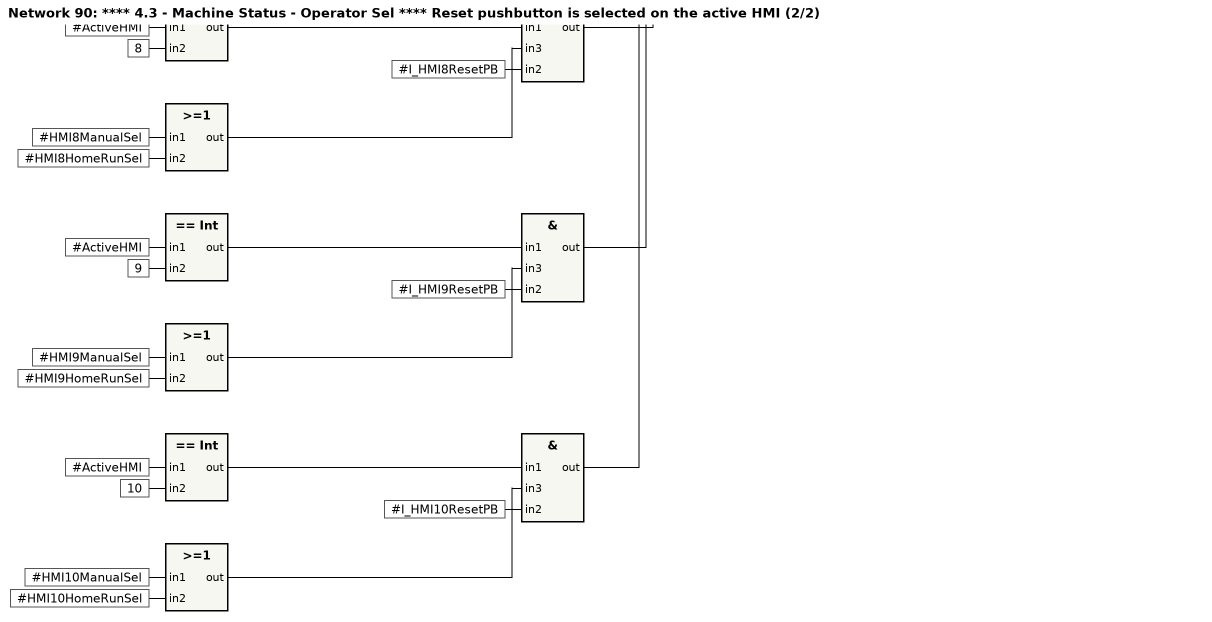
   #O_PBResetSel := (((#ActiveHMI = 1) AND (#HMI1ManualSel OR #HMI1HomeRunSel) AND #I_HMI1ResetPB) OR ((#ActiveHMI = 2) AND (#HMI2ManualSel OR #HMI2HomeRunSel) AND #I_HMI2ResetPB) OR ((#ActiveHMI = 3) AND (#HMI3ManualSel OR #HMI3HomeRunSel) AND #I_HMI3ResetPB) OR ((#ActiveHMI = 4) AND (#HMI4ManualSel OR #HMI4HomeRunSel) AND #I_HMI4ResetPB) OR ((#ActiveHMI = 5) AND (#HMI5ManualSel OR #HMI5HomeRunSel) AND #I_HMI5ResetPB) OR ((#ActiveHMI = 6) AND (#HMI6ManualSel OR #HMI6HomeRunSel) AND #I_HMI6ResetPB) OR ((#ActiveHMI = 7) AND (#HMI7ManualSel OR #HMI7HomeRunSel) AND #I_HMI7ResetPB) OR ((#ActiveHMI = 8) AND (#HMI8ManualSel OR #HMI8HomeRunSel) AND #I_HMI8ResetPB) OR ((#ActiveHMI = 9) AND (#HMI9ManualSel OR #HMI9HomeRunSel) AND #I_HMI9ResetPB) OR ((#ActiveHMI = 10) AND (#HMI10ManualSel OR #HMI10HomeRunSel) AND #I_HMI10ResetPB)) AND NOT #AllHmiAutoSel;
   #PBResetSel := #O_PBResetSel;
   #IO_Modes.LModeSelector.PBResetSel := #O_PBResetSel;
END_REGION

REGION Network 91: **** 4.3 - Machine Status - Operator Sel **** Homerun Redo is selected
   // Homerun Redo is selected
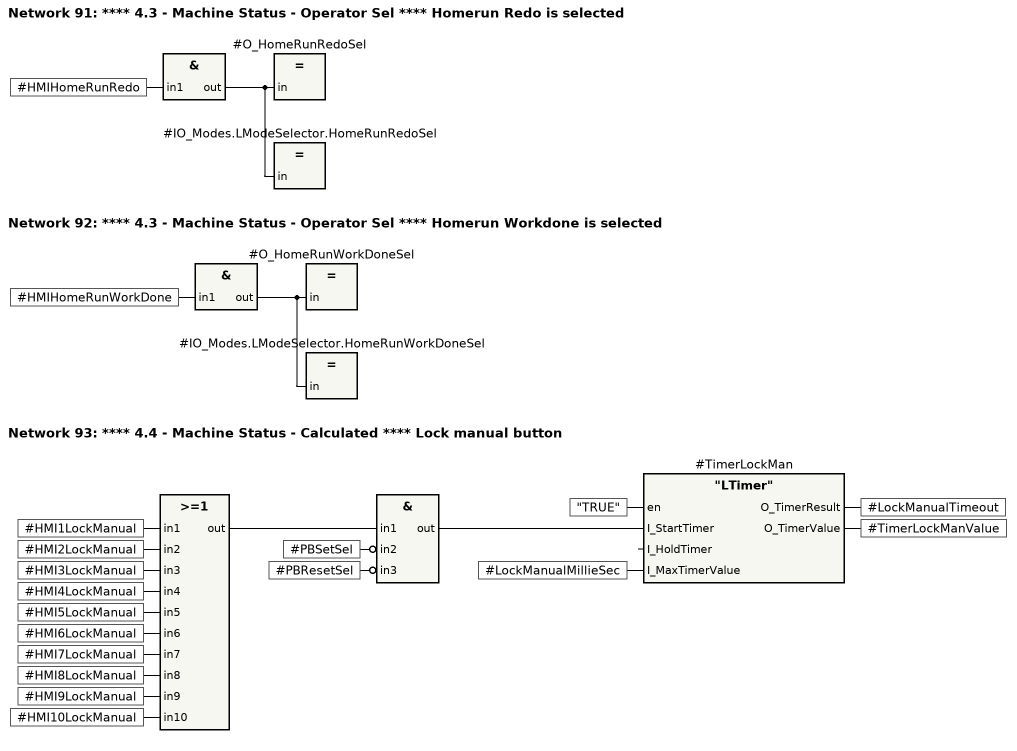
   #O_HomeRunRedoSel := #HMIHomeRunRedo;
   #IO_Modes.LModeSelector.HomeRunRedoSel := #HMIHomeRunRedo;
END_REGION

REGION Network 92: **** 4.3 - Machine Status - Operator Sel **** Homerun Workdone is selected
   // Homerun Workdone is selected
   #O_HomeRunWorkDoneSel := #HMIHomeRunWorkDone;
   #IO_Modes.LModeSelector.HomeRunWorkDoneSel := #HMIHomeRunWorkDone;
END_REGION

REGION Network 93: **** 4.4 - Machine Status - Calculated **** Lock manual button
   // Lock manual button
   IF "TRUE" THEN
       #TimerLockMan(I_StartTimer := (#HMI1LockManual OR #HMI2LockManual OR #HMI3LockManual OR #HMI4LockManual OR #HMI5LockManual OR #HMI6LockManual OR #HMI7LockManual OR #HMI8LockManual OR #HMI9LockManual OR #HMI10LockManual) AND NOT #PBSetSel AND NOT #PBResetSel,   // "LTimer"
                     I_MaxTimerValue := #LockManualMillieSec,
                     O_TimerResult => #LockManualTimeout,
                     O_TimerValue => #TimerLockManValue);
   END_IF;
END_REGION

REGION Network 94: **** 4.5 - Machine Status - Modes **** Auto is selected on all HMI
   // Auto is selected on all HMI
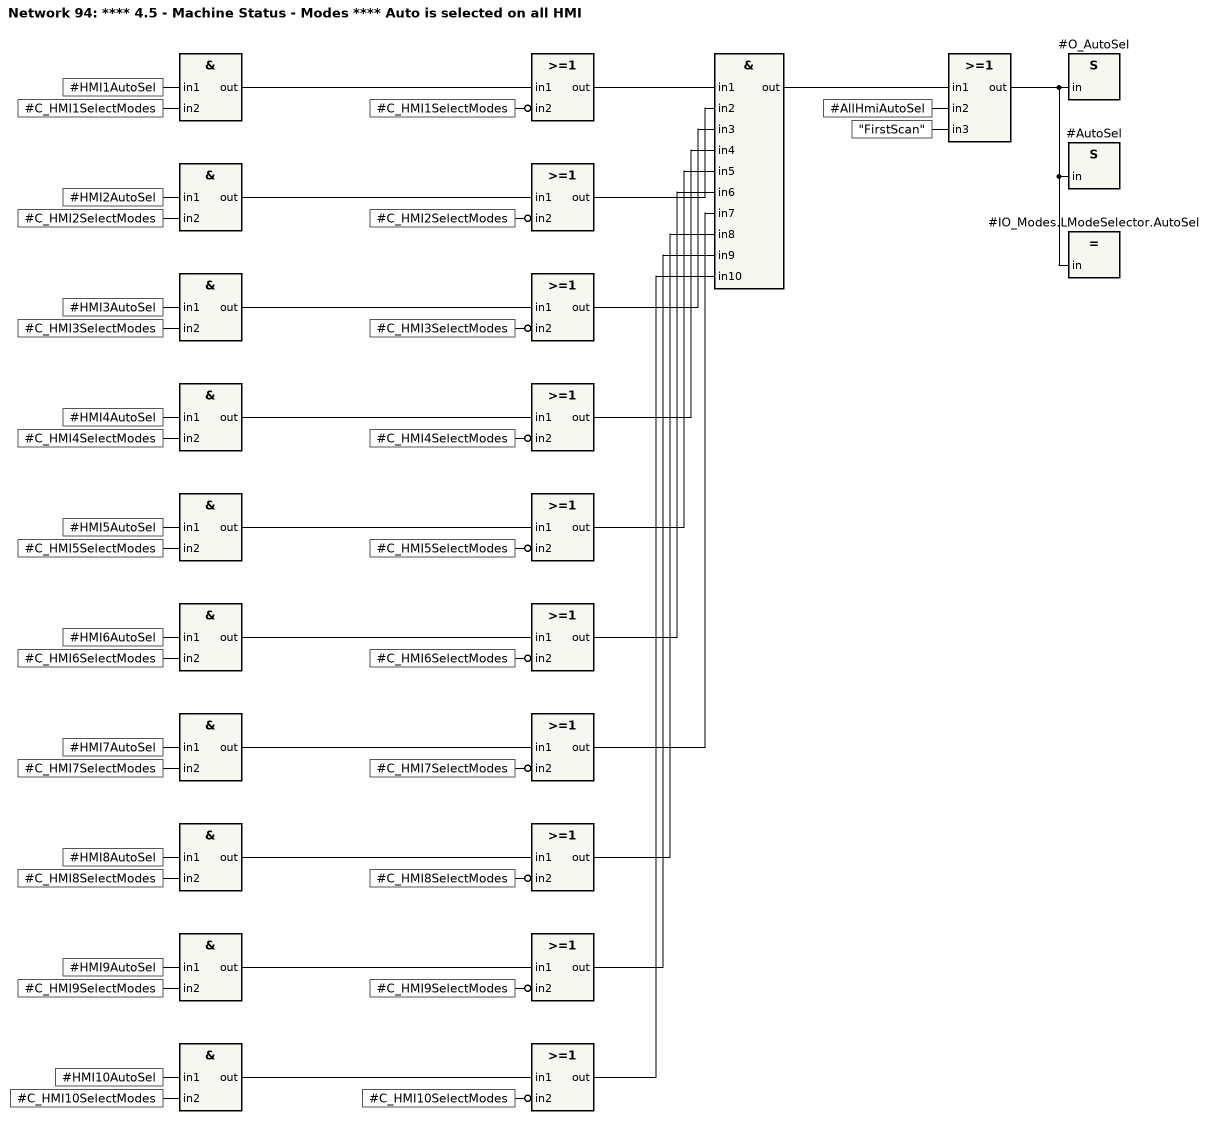
   #_w1 := (((#HMI1AutoSel AND #C_HMI1SelectModes) OR NOT #C_HMI1SelectModes) AND ((#HMI2AutoSel AND #C_HMI2SelectModes) OR NOT #C_HMI2SelectModes) AND ((#HMI3AutoSel AND #C_HMI3SelectModes) OR NOT #C_HMI3SelectModes) AND ((#HMI4AutoSel AND #C_HMI4SelectModes) OR NOT #C_HMI4SelectModes) AND ((#HMI5AutoSel AND #C_HMI5SelectModes) OR NOT #C_HMI5SelectModes) AND ((#HMI6AutoSel AND #C_HMI6SelectModes) OR NOT #C_HMI6SelectModes) AND ((#HMI7AutoSel AND #C_HMI7SelectModes) OR NOT #C_HMI7SelectModes) AND ((#HMI8AutoSel AND #C_HMI8SelectModes) OR NOT #C_HMI8SelectModes) AND ((#HMI9AutoSel AND #C_HMI9SelectModes) OR NOT #C_HMI9SelectModes) AND ((#HMI10AutoSel AND #C_HMI10SelectModes) OR NOT #C_HMI10SelectModes)) OR #AllHmiAutoSel OR "FirstScan";
   IF #_w1 THEN
       #O_AutoSel := TRUE;
       #AutoSel := TRUE;
   END_IF;
   #IO_Modes.LModeSelector.AutoSel := #_w1;
END_REGION

REGION Network 95: **** 4.5 - Machine Status - Modes **** Reset Auto is selected on all HMI
   // Reset Auto is selected on all HMI
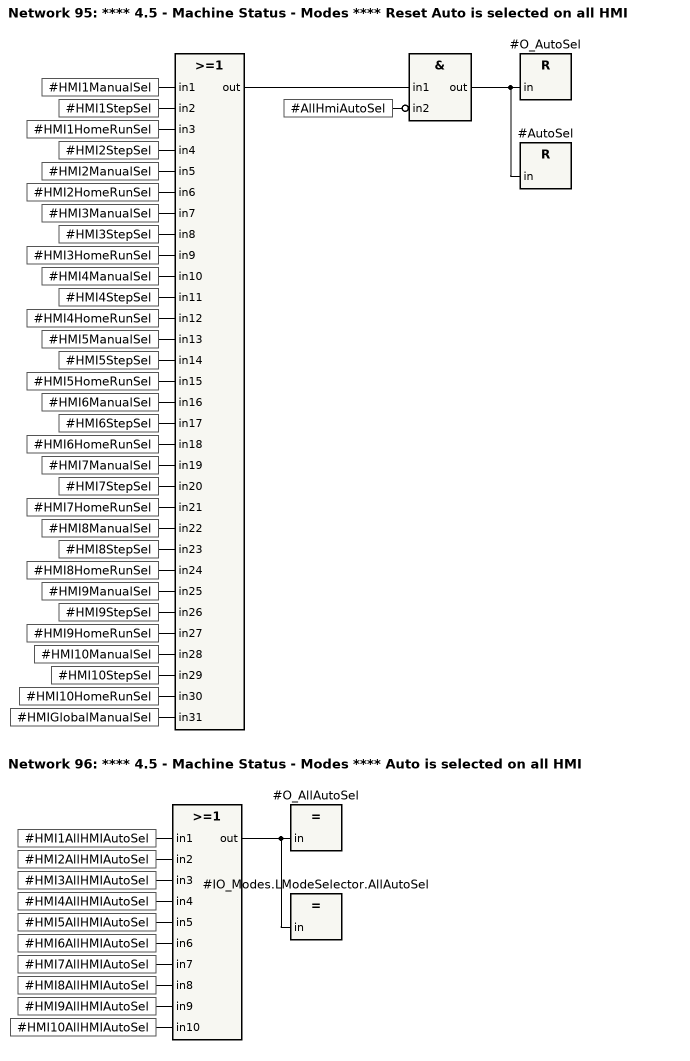
   IF (#HMI1ManualSel OR #HMI1StepSel OR #HMI1HomeRunSel OR #HMI2StepSel OR #HMI2ManualSel OR #HMI2HomeRunSel OR #HMI3ManualSel OR #HMI3StepSel OR #HMI3HomeRunSel OR #HMI4ManualSel OR #HMI4StepSel OR #HMI4HomeRunSel OR #HMI5ManualSel OR #HMI5StepSel OR #HMI5HomeRunSel OR #HMI6ManualSel OR #HMI6StepSel OR #HMI6HomeRunSel OR #HMI7ManualSel OR #HMI7StepSel OR #HMI7HomeRunSel OR #HMI8ManualSel OR #HMI8StepSel OR #HMI8HomeRunSel OR #HMI9ManualSel OR #HMI9StepSel OR #HMI9HomeRunSel OR #HMI10ManualSel OR #HMI10StepSel OR #HMI10HomeRunSel OR #HMIGlobalManualSel) AND NOT #AllHmiAutoSel THEN
       #O_AutoSel := FALSE;
       #AutoSel := FALSE;
   END_IF;
END_REGION

REGION Network 96: **** 4.5 - Machine Status - Modes **** Auto is selected on all HMI
   // Auto is selected on all HMI
   #O_AllAutoSel := #HMI1AllHMIAutoSel OR #HMI2AllHMIAutoSel OR #HMI3AllHMIAutoSel OR #HMI4AllHMIAutoSel OR #HMI5AllHMIAutoSel OR #HMI6AllHMIAutoSel OR #HMI7AllHMIAutoSel OR #HMI8AllHMIAutoSel OR #HMI9AllHMIAutoSel OR #HMI10AllHMIAutoSel;
   #IO_Modes.LModeSelector.AllAutoSel := #O_AllAutoSel;
END_REGION

REGION Network 97: **** 4.5 - Machine Status - Modes **** Step is selected on one HMI
   // Step is selected on one HMI
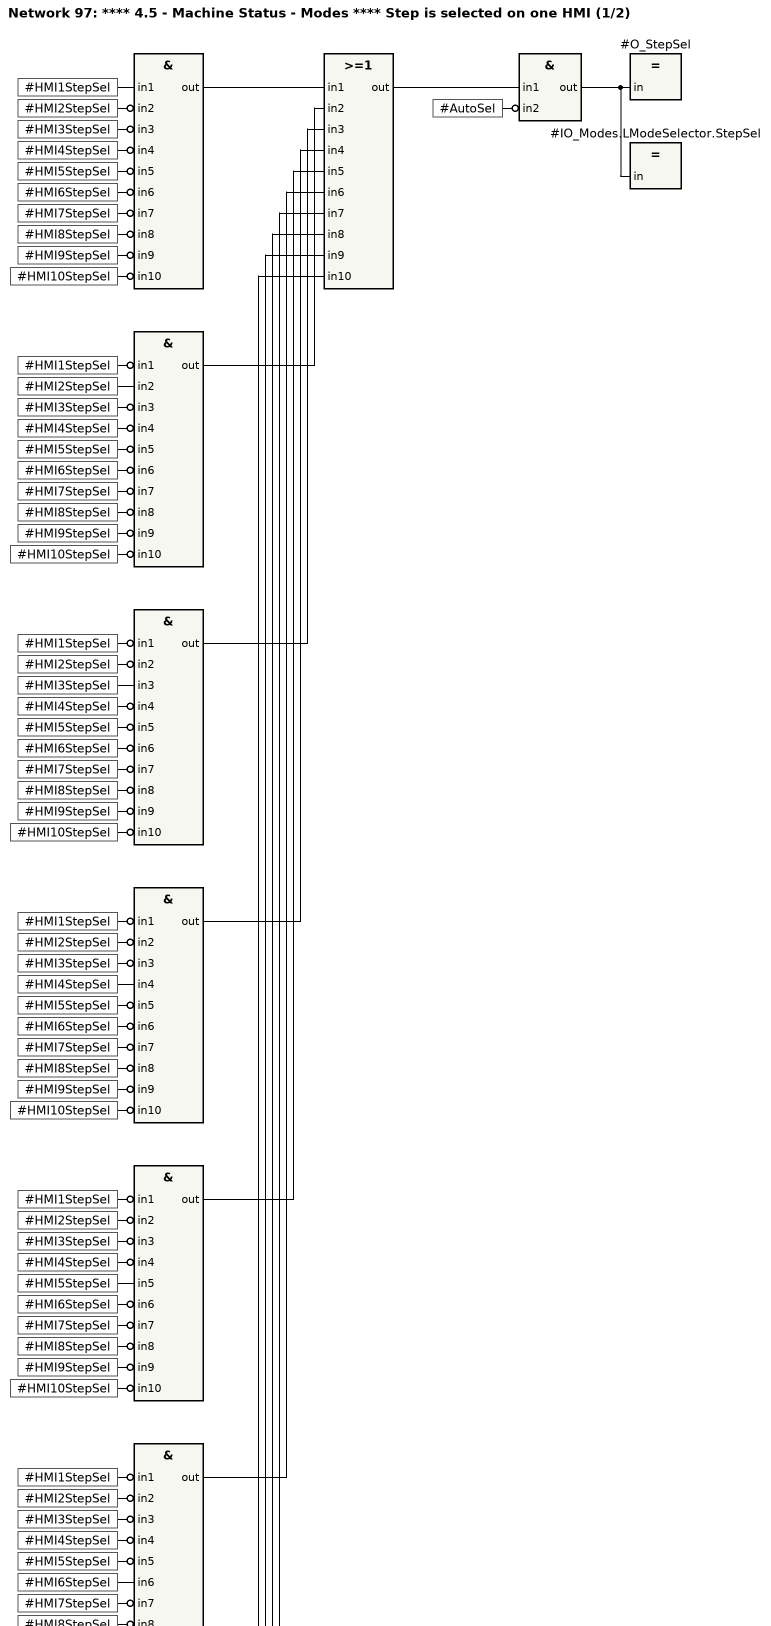
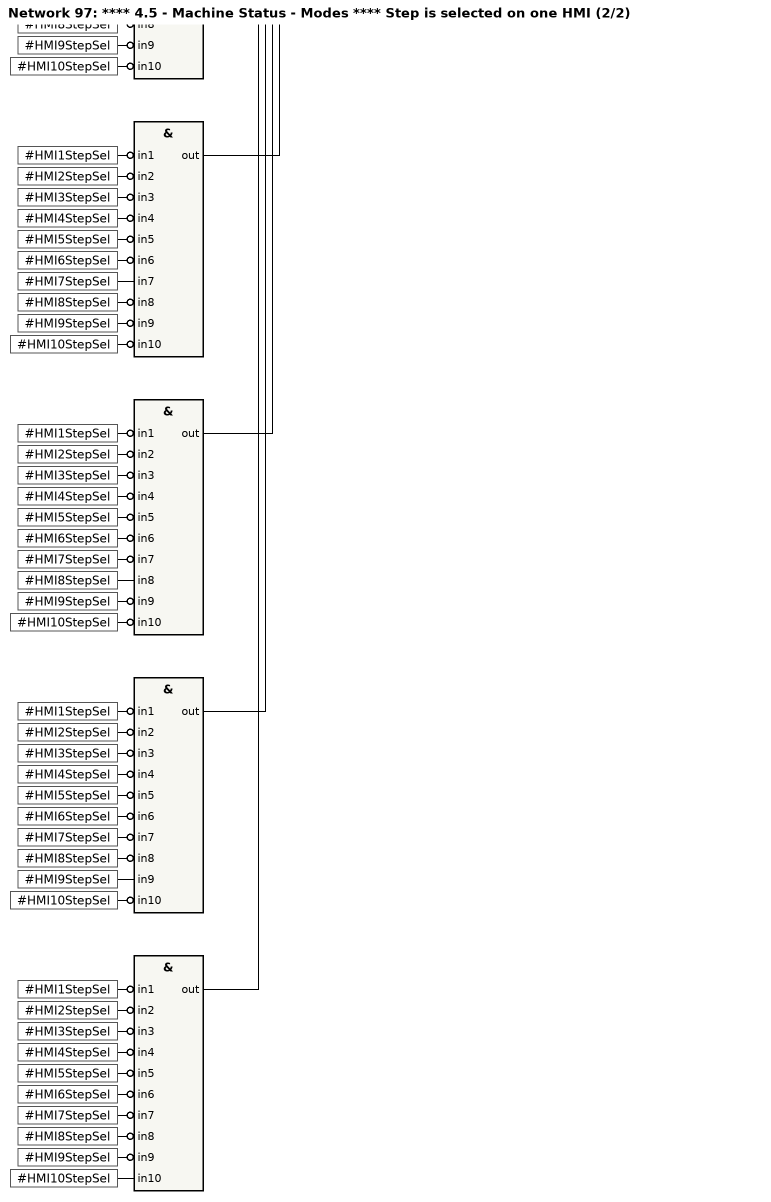
   #O_StepSel := ((#HMI1StepSel AND NOT #HMI2StepSel AND NOT #HMI3StepSel AND NOT #HMI4StepSel AND NOT #HMI5StepSel AND NOT #HMI6StepSel AND NOT #HMI7StepSel AND NOT #HMI8StepSel AND NOT #HMI9StepSel AND NOT #HMI10StepSel) OR (NOT #HMI1StepSel AND #HMI2StepSel AND NOT #HMI3StepSel AND NOT #HMI4StepSel AND NOT #HMI5StepSel AND NOT #HMI6StepSel AND NOT #HMI7StepSel AND NOT #HMI8StepSel AND NOT #HMI9StepSel AND NOT #HMI10StepSel) OR (NOT #HMI1StepSel AND NOT #HMI2StepSel AND #HMI3StepSel AND NOT #HMI4StepSel AND NOT #HMI5StepSel AND NOT #HMI6StepSel AND NOT #HMI7StepSel AND NOT #HMI8StepSel AND NOT #HMI9StepSel AND NOT #HMI10StepSel) OR (NOT #HMI1StepSel AND NOT #HMI2StepSel AND NOT #HMI3StepSel AND #HMI4StepSel AND NOT #HMI5StepSel AND NOT #HMI6StepSel AND NOT #HMI7StepSel AND NOT #HMI8StepSel AND NOT #HMI9StepSel AND NOT #HMI10StepSel) OR (NOT #HMI1StepSel AND NOT #HMI2StepSel AND NOT #HMI3StepSel AND NOT #HMI4StepSel AND #HMI5StepSel AND NOT #HMI6StepSel AND NOT #HMI7StepSel AND NOT #HMI8StepSel AND NOT #HMI9StepSel AND NOT #HMI10StepSel) OR (NOT #HMI1StepSel AND NOT #HMI2StepSel AND NOT #HMI3StepSel AND NOT #HMI4StepSel AND NOT #HMI5StepSel AND #HMI6StepSel AND NOT #HMI7StepSel AND NOT #HMI8StepSel AND NOT #HMI9StepSel AND NOT #HMI10StepSel) OR (NOT #HMI1StepSel AND NOT #HMI2StepSel AND NOT #HMI3StepSel AND NOT #HMI4StepSel AND NOT #HMI5StepSel AND NOT #HMI6StepSel AND #HMI7StepSel AND NOT #HMI8StepSel AND NOT #HMI9StepSel AND NOT #HMI10StepSel) OR (NOT #HMI1StepSel AND NOT #HMI2StepSel AND NOT #HMI3StepSel AND NOT #HMI4StepSel AND NOT #HMI5StepSel AND NOT #HMI6StepSel AND NOT #HMI7StepSel AND #HMI8StepSel AND NOT #HMI9StepSel AND NOT #HMI10StepSel) OR (NOT #HMI1StepSel AND NOT #HMI2StepSel AND NOT #HMI3StepSel AND NOT #HMI4StepSel AND NOT #HMI5StepSel AND NOT #HMI6StepSel AND NOT #HMI7StepSel AND NOT #HMI8StepSel AND #HMI9StepSel AND NOT #HMI10StepSel) OR (NOT #HMI1StepSel AND NOT #HMI2StepSel AND NOT #HMI3StepSel AND NOT #HMI4StepSel AND NOT #HMI5StepSel AND NOT #HMI6StepSel AND NOT #HMI7StepSel AND NOT #HMI8StepSel AND NOT #HMI9StepSel AND #HMI10StepSel)) AND NOT #AutoSel;
   #IO_Modes.LModeSelector.StepSel := #O_StepSel;
END_REGION

REGION Network 98: **** 4.5 - Machine Status - Modes **** Homerun is selected on one HMI
   // Homerun is selected on one HMI
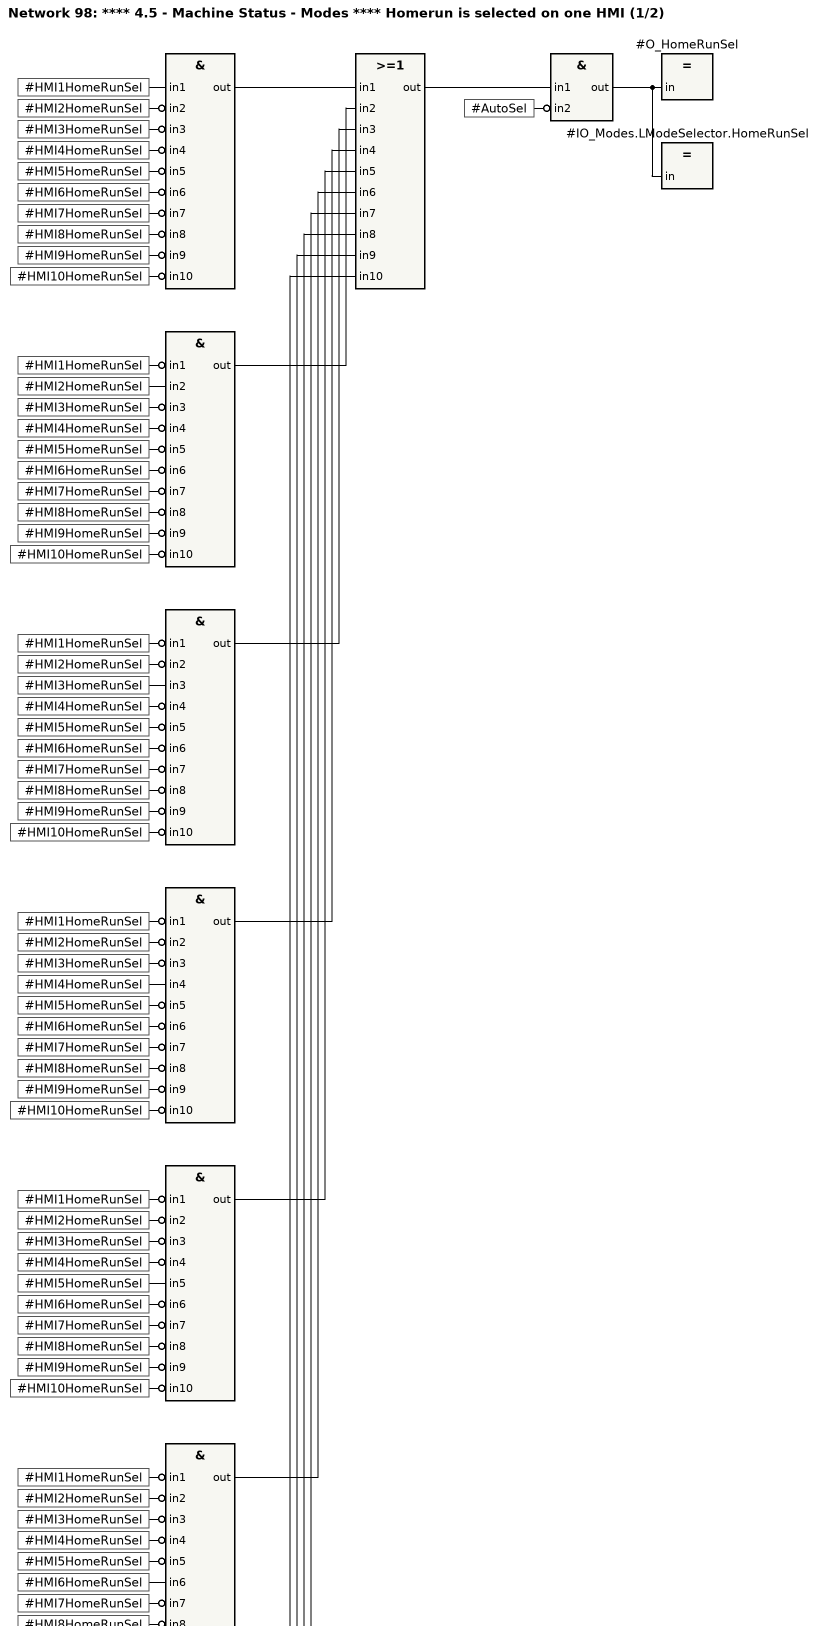
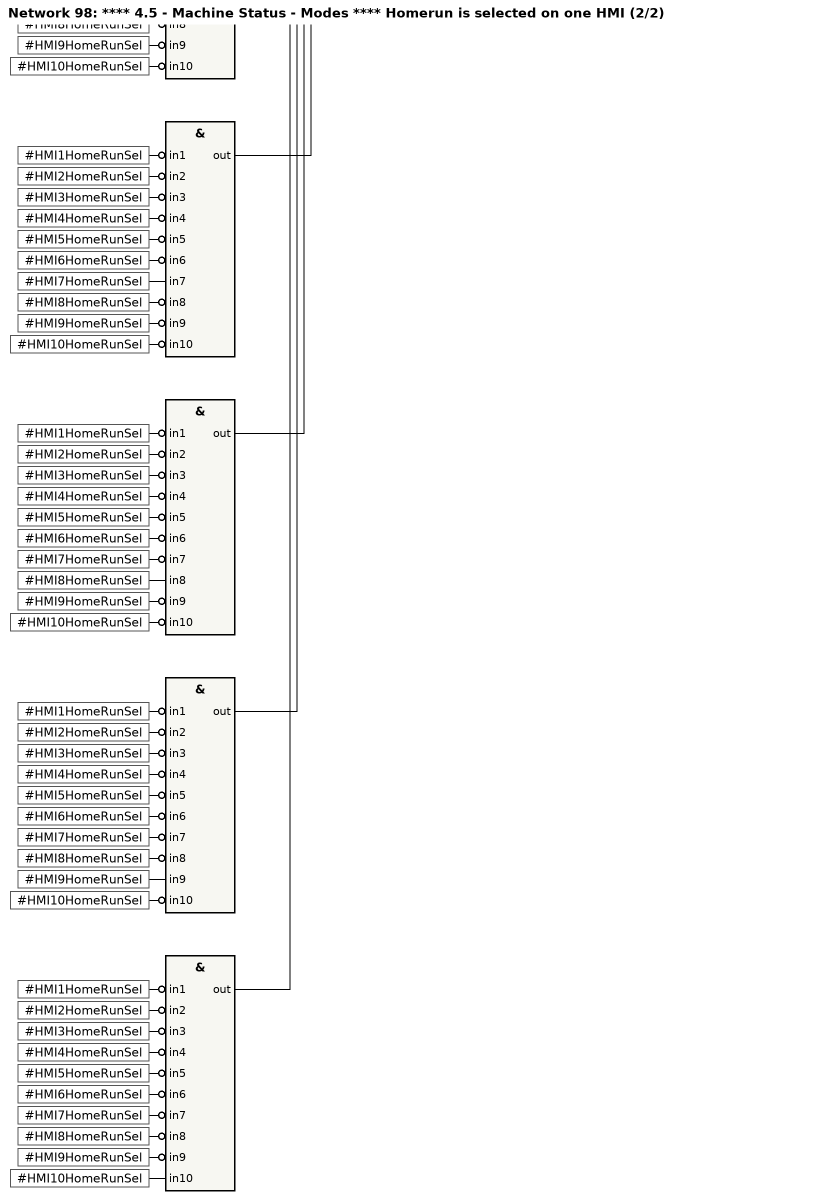
   #O_HomeRunSel := ((#HMI1HomeRunSel AND NOT #HMI2HomeRunSel AND NOT #HMI3HomeRunSel AND NOT #HMI4HomeRunSel AND NOT #HMI5HomeRunSel AND NOT #HMI6HomeRunSel AND NOT #HMI7HomeRunSel AND NOT #HMI8HomeRunSel AND NOT #HMI9HomeRunSel AND NOT #HMI10HomeRunSel) OR (NOT #HMI1HomeRunSel AND #HMI2HomeRunSel AND NOT #HMI3HomeRunSel AND NOT #HMI4HomeRunSel AND NOT #HMI5HomeRunSel AND NOT #HMI6HomeRunSel AND NOT #HMI7HomeRunSel AND NOT #HMI8HomeRunSel AND NOT #HMI9HomeRunSel AND NOT #HMI10HomeRunSel) OR (NOT #HMI1HomeRunSel AND NOT #HMI2HomeRunSel AND #HMI3HomeRunSel AND NOT #HMI4HomeRunSel AND NOT #HMI5HomeRunSel AND NOT #HMI6HomeRunSel AND NOT #HMI7HomeRunSel AND NOT #HMI8HomeRunSel AND NOT #HMI9HomeRunSel AND NOT #HMI10HomeRunSel) OR (NOT #HMI1HomeRunSel AND NOT #HMI2HomeRunSel AND NOT #HMI3HomeRunSel AND #HMI4HomeRunSel AND NOT #HMI5HomeRunSel AND NOT #HMI6HomeRunSel AND NOT #HMI7HomeRunSel AND NOT #HMI8HomeRunSel AND NOT #HMI9HomeRunSel AND NOT #HMI10HomeRunSel) OR (NOT #HMI1HomeRunSel AND NOT #HMI2HomeRunSel AND NOT #HMI3HomeRunSel AND NOT #HMI4HomeRunSel AND #HMI5HomeRunSel AND NOT #HMI6HomeRunSel AND NOT #HMI7HomeRunSel AND NOT #HMI8HomeRunSel AND NOT #HMI9HomeRunSel AND NOT #HMI10HomeRunSel) OR (NOT #HMI1HomeRunSel AND NOT #HMI2HomeRunSel AND NOT #HMI3HomeRunSel AND NOT #HMI4HomeRunSel AND NOT #HMI5HomeRunSel AND #HMI6HomeRunSel AND NOT #HMI7HomeRunSel AND NOT #HMI8HomeRunSel AND NOT #HMI9HomeRunSel AND NOT #HMI10HomeRunSel) OR (NOT #HMI1HomeRunSel AND NOT #HMI2HomeRunSel AND NOT #HMI3HomeRunSel AND NOT #HMI4HomeRunSel AND NOT #HMI5HomeRunSel AND NOT #HMI6HomeRunSel AND #HMI7HomeRunSel AND NOT #HMI8HomeRunSel AND NOT #HMI9HomeRunSel AND NOT #HMI10HomeRunSel) OR (NOT #HMI1HomeRunSel AND NOT #HMI2HomeRunSel AND NOT #HMI3HomeRunSel AND NOT #HMI4HomeRunSel AND NOT #HMI5HomeRunSel AND NOT #HMI6HomeRunSel AND NOT #HMI7HomeRunSel AND #HMI8HomeRunSel AND NOT #HMI9HomeRunSel AND NOT #HMI10HomeRunSel) OR (NOT #HMI1HomeRunSel AND NOT #HMI2HomeRunSel AND NOT #HMI3HomeRunSel AND NOT #HMI4HomeRunSel AND NOT #HMI5HomeRunSel AND NOT #HMI6HomeRunSel AND NOT #HMI7HomeRunSel AND NOT #HMI8HomeRunSel AND #HMI9HomeRunSel AND NOT #HMI10HomeRunSel) OR (NOT #HMI1HomeRunSel AND NOT #HMI2HomeRunSel AND NOT #HMI3HomeRunSel AND NOT #HMI4HomeRunSel AND NOT #HMI5HomeRunSel AND NOT #HMI6HomeRunSel AND NOT #HMI7HomeRunSel AND NOT #HMI8HomeRunSel AND NOT #HMI9HomeRunSel AND #HMI10HomeRunSel)) AND NOT #AutoSel;
   #IO_Modes.LModeSelector.HomeRunSel := #O_HomeRunSel;
END_REGION

REGION Network 99: **** 4.5 - Machine Status - Modes **** Reset activ HMI
   // Reset activ HMI
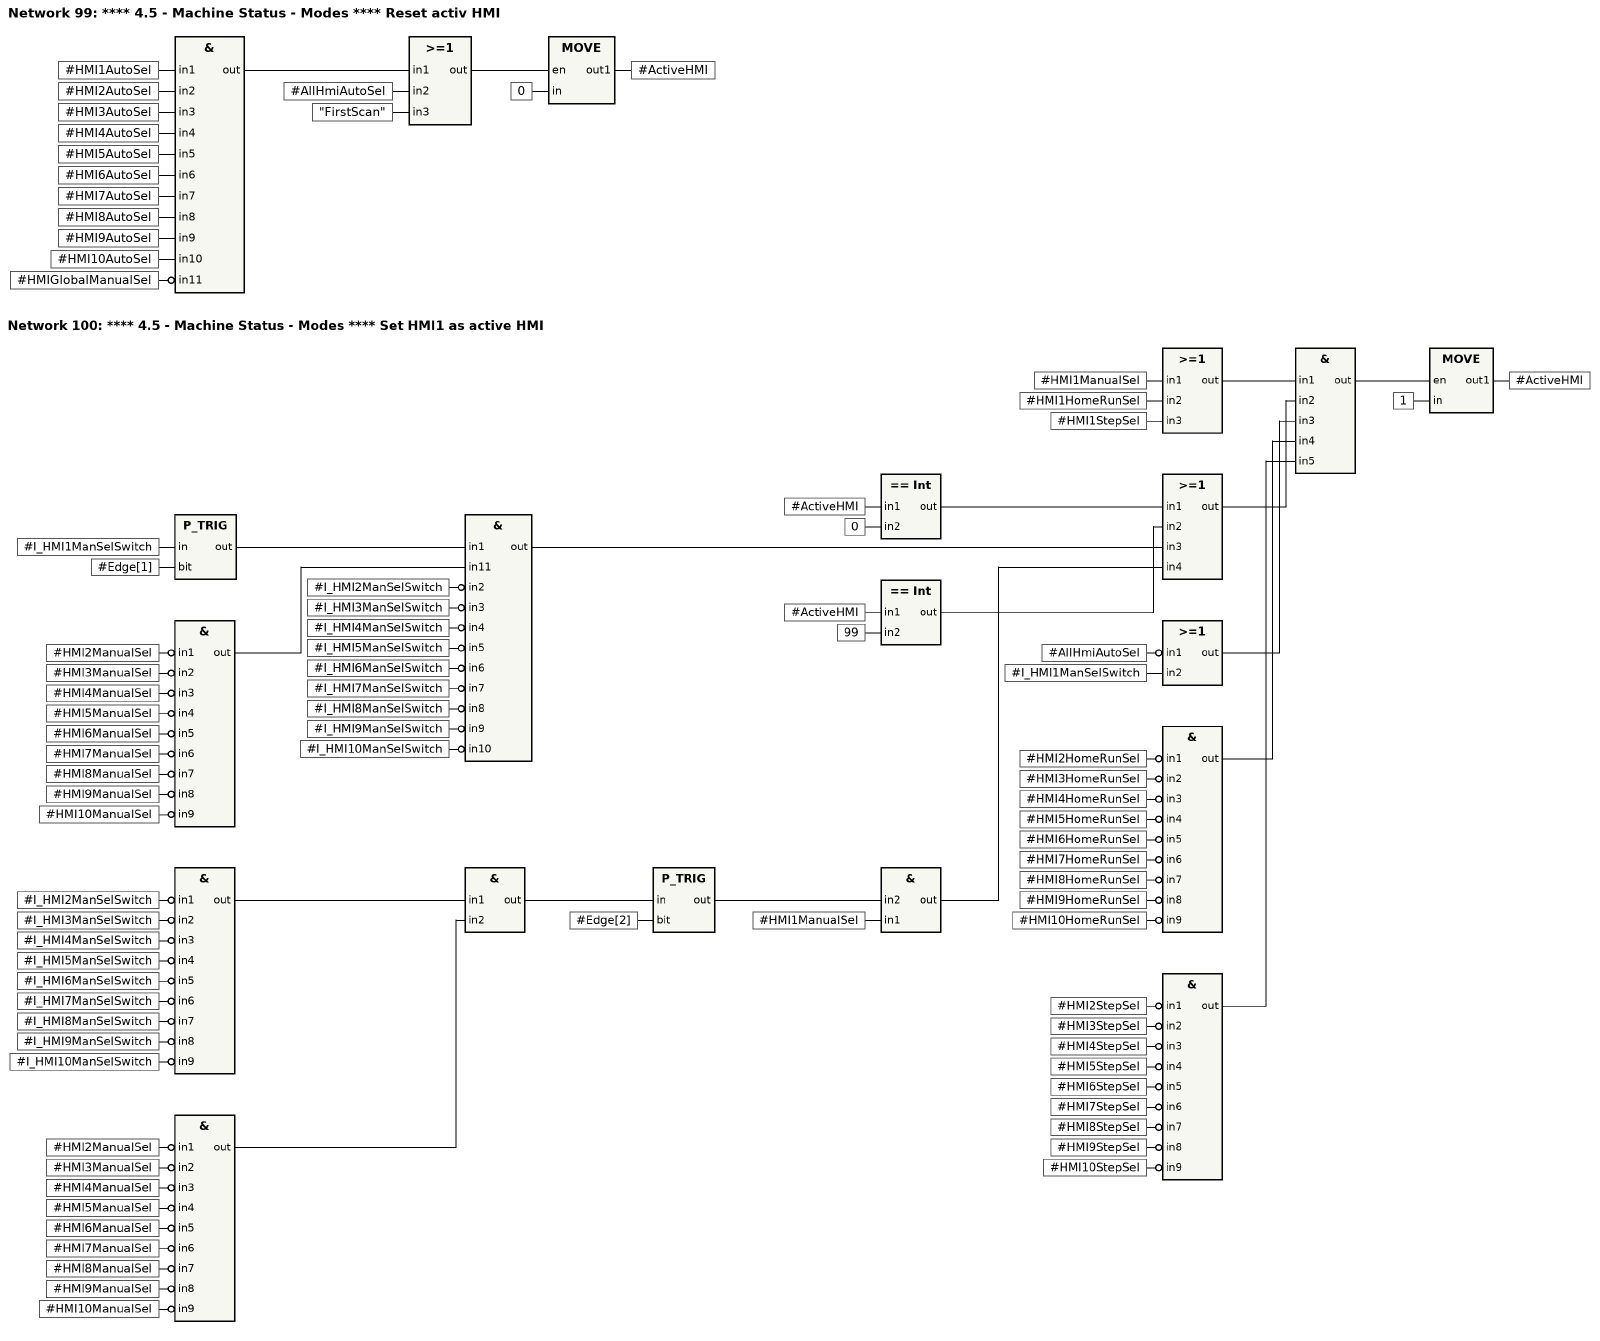
   IF (#HMI1AutoSel AND #HMI2AutoSel AND #HMI3AutoSel AND #HMI4AutoSel AND #HMI5AutoSel AND #HMI6AutoSel AND #HMI7AutoSel AND #HMI8AutoSel AND #HMI9AutoSel AND #HMI10AutoSel AND NOT #HMIGlobalManualSel) OR #AllHmiAutoSel OR "FirstScan" THEN
       #ActiveHMI := 0;
   END_IF;
END_REGION

REGION Network 100: **** 4.5 - Machine Status - Modes **** Set HMI1 as active HMI
   // Set HMI1 as active HMI
   #_w1 := #I_HMI1ManSelSwitch AND NOT #Edge[1];   // rising edge
   #Edge[1] := #I_HMI1ManSelSwitch;
   #_w2 := NOT #I_HMI2ManSelSwitch AND NOT #I_HMI3ManSelSwitch AND NOT #I_HMI4ManSelSwitch AND NOT #I_HMI5ManSelSwitch AND NOT #I_HMI6ManSelSwitch AND NOT #I_HMI7ManSelSwitch AND NOT #I_HMI8ManSelSwitch AND NOT #I_HMI9ManSelSwitch AND NOT #I_HMI10ManSelSwitch AND NOT #HMI2ManualSel AND NOT #HMI3ManualSel AND NOT #HMI4ManualSel AND NOT #HMI5ManualSel AND NOT #HMI6ManualSel AND NOT #HMI7ManualSel AND NOT #HMI8ManualSel AND NOT #HMI9ManualSel AND NOT #HMI10ManualSel;
   #_w3 := #_w2 AND NOT #Edge[2];   // rising edge
   #Edge[2] := #_w2;
   IF (#HMI1ManualSel OR #HMI1HomeRunSel OR #HMI1StepSel) AND ((#ActiveHMI = 0) OR (#ActiveHMI = 99) OR (#_w1 AND NOT #HMI2ManualSel AND NOT #HMI3ManualSel AND NOT #HMI4ManualSel AND NOT #HMI5ManualSel AND NOT #HMI6ManualSel AND NOT #HMI7ManualSel AND NOT #HMI8ManualSel AND NOT #HMI9ManualSel AND NOT #HMI10ManualSel AND NOT #I_HMI2ManSelSwitch AND NOT #I_HMI3ManSelSwitch AND NOT #I_HMI4ManSelSwitch AND NOT #I_HMI5ManSelSwitch AND NOT #I_HMI6ManSelSwitch AND NOT #I_HMI7ManSelSwitch AND NOT #I_HMI8ManSelSwitch AND NOT #I_HMI9ManSelSwitch AND NOT #I_HMI10ManSelSwitch) OR (#_w3 AND #HMI1ManualSel)) AND (NOT #AllHmiAutoSel OR #I_HMI1ManSelSwitch) AND NOT #HMI2HomeRunSel AND NOT #HMI3HomeRunSel AND NOT #HMI4HomeRunSel AND NOT #HMI5HomeRunSel AND NOT #HMI6HomeRunSel AND NOT #HMI7HomeRunSel AND NOT #HMI8HomeRunSel AND NOT #HMI9HomeRunSel AND NOT #HMI10HomeRunSel AND NOT #HMI2StepSel AND NOT #HMI3StepSel AND NOT #HMI4StepSel AND NOT #HMI5StepSel AND NOT #HMI6StepSel AND NOT #HMI7StepSel AND NOT #HMI8StepSel AND NOT #HMI9StepSel AND NOT #HMI10StepSel THEN
       #ActiveHMI := 1;
   END_IF;
END_REGION

REGION Network 101: **** 4.5 - Machine Status - Modes **** Set HMI2 as active HMI
   // Set HMI2 as active HMI
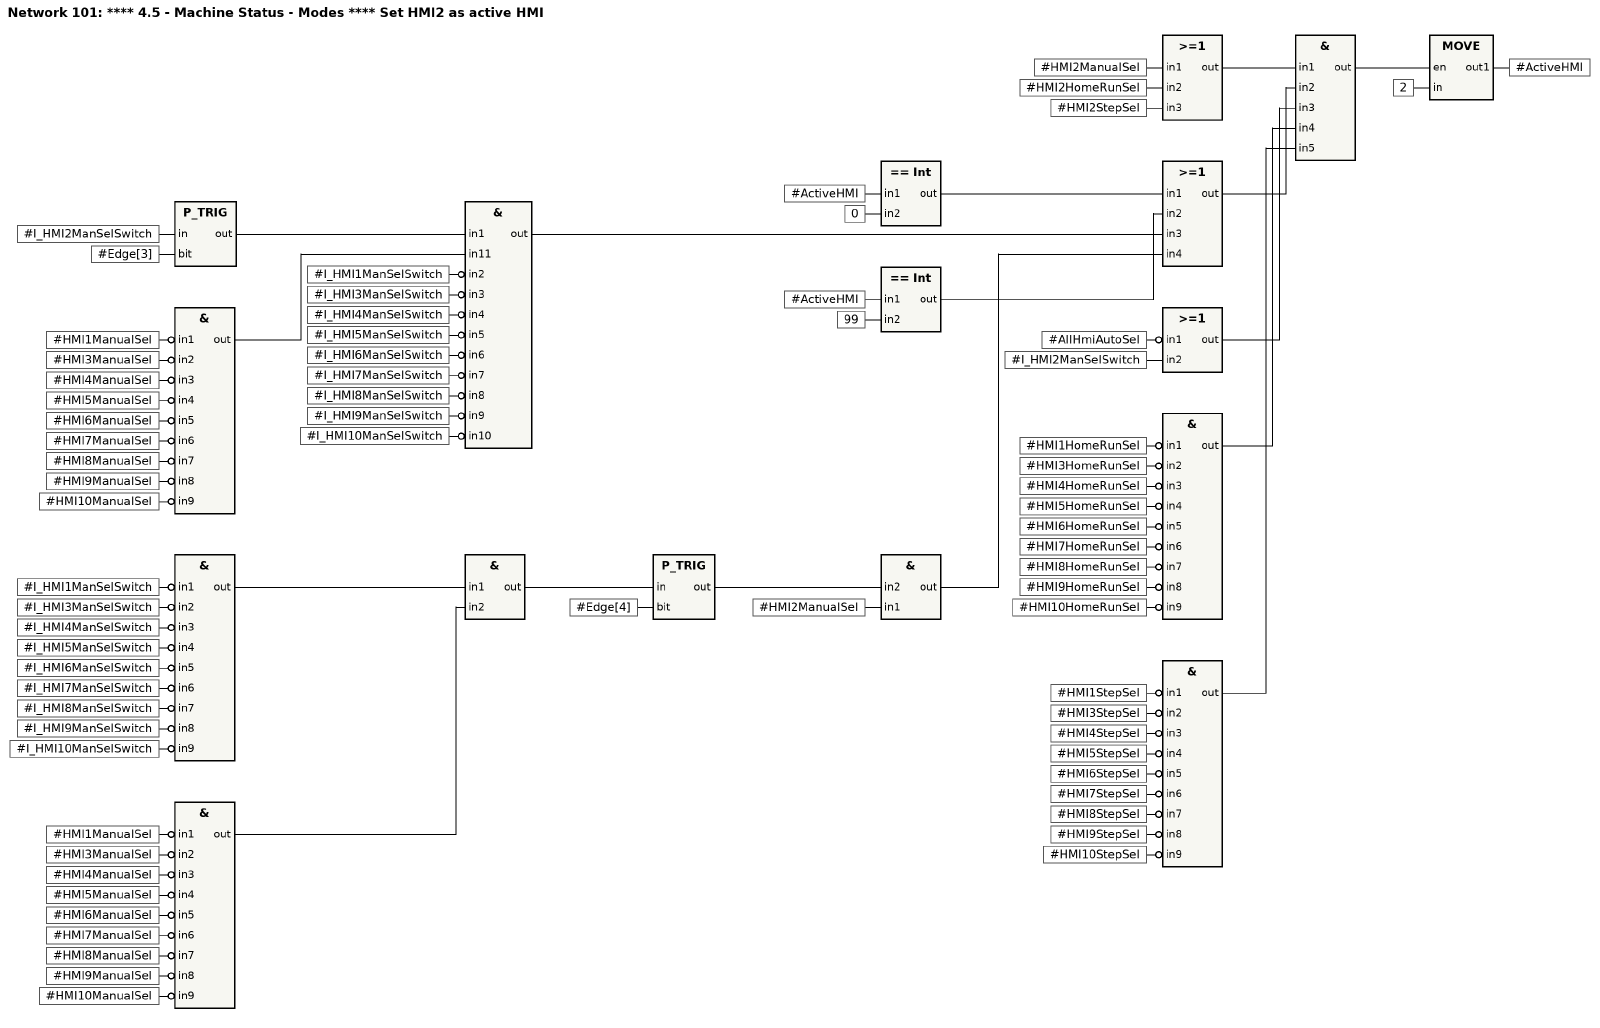
   #_w1 := #I_HMI2ManSelSwitch AND NOT #Edge[3];   // rising edge
   #Edge[3] := #I_HMI2ManSelSwitch;
   #_w2 := NOT #I_HMI1ManSelSwitch AND NOT #I_HMI3ManSelSwitch AND NOT #I_HMI4ManSelSwitch AND NOT #I_HMI5ManSelSwitch AND NOT #I_HMI6ManSelSwitch AND NOT #I_HMI7ManSelSwitch AND NOT #I_HMI8ManSelSwitch AND NOT #I_HMI9ManSelSwitch AND NOT #I_HMI10ManSelSwitch AND NOT #HMI1ManualSel AND NOT #HMI3ManualSel AND NOT #HMI4ManualSel AND NOT #HMI5ManualSel AND NOT #HMI6ManualSel AND NOT #HMI7ManualSel AND NOT #HMI8ManualSel AND NOT #HMI9ManualSel AND NOT #HMI10ManualSel;
   #_w3 := #_w2 AND NOT #Edge[4];   // rising edge
   #Edge[4] := #_w2;
   IF (#HMI2ManualSel OR #HMI2HomeRunSel OR #HMI2StepSel) AND ((#ActiveHMI = 0) OR (#ActiveHMI = 99) OR (#_w1 AND NOT #HMI1ManualSel AND NOT #HMI3ManualSel AND NOT #HMI4ManualSel AND NOT #HMI5ManualSel AND NOT #HMI6ManualSel AND NOT #HMI7ManualSel AND NOT #HMI8ManualSel AND NOT #HMI9ManualSel AND NOT #HMI10ManualSel AND NOT #I_HMI1ManSelSwitch AND NOT #I_HMI3ManSelSwitch AND NOT #I_HMI4ManSelSwitch AND NOT #I_HMI5ManSelSwitch AND NOT #I_HMI6ManSelSwitch AND NOT #I_HMI7ManSelSwitch AND NOT #I_HMI8ManSelSwitch AND NOT #I_HMI9ManSelSwitch AND NOT #I_HMI10ManSelSwitch) OR (#_w3 AND #HMI2ManualSel)) AND (NOT #AllHmiAutoSel OR #I_HMI2ManSelSwitch) AND NOT #HMI1HomeRunSel AND NOT #HMI3HomeRunSel AND NOT #HMI4HomeRunSel AND NOT #HMI5HomeRunSel AND NOT #HMI6HomeRunSel AND NOT #HMI7HomeRunSel AND NOT #HMI8HomeRunSel AND NOT #HMI9HomeRunSel AND NOT #HMI10HomeRunSel AND NOT #HMI1StepSel AND NOT #HMI3StepSel AND NOT #HMI4StepSel AND NOT #HMI5StepSel AND NOT #HMI6StepSel AND NOT #HMI7StepSel AND NOT #HMI8StepSel AND NOT #HMI9StepSel AND NOT #HMI10StepSel THEN
       #ActiveHMI := 2;
   END_IF;
END_REGION

REGION Network 102: **** 4.5 - Machine Status - Modes **** Set HMI3 as active HMI
   // Set HMI3 as active HMI
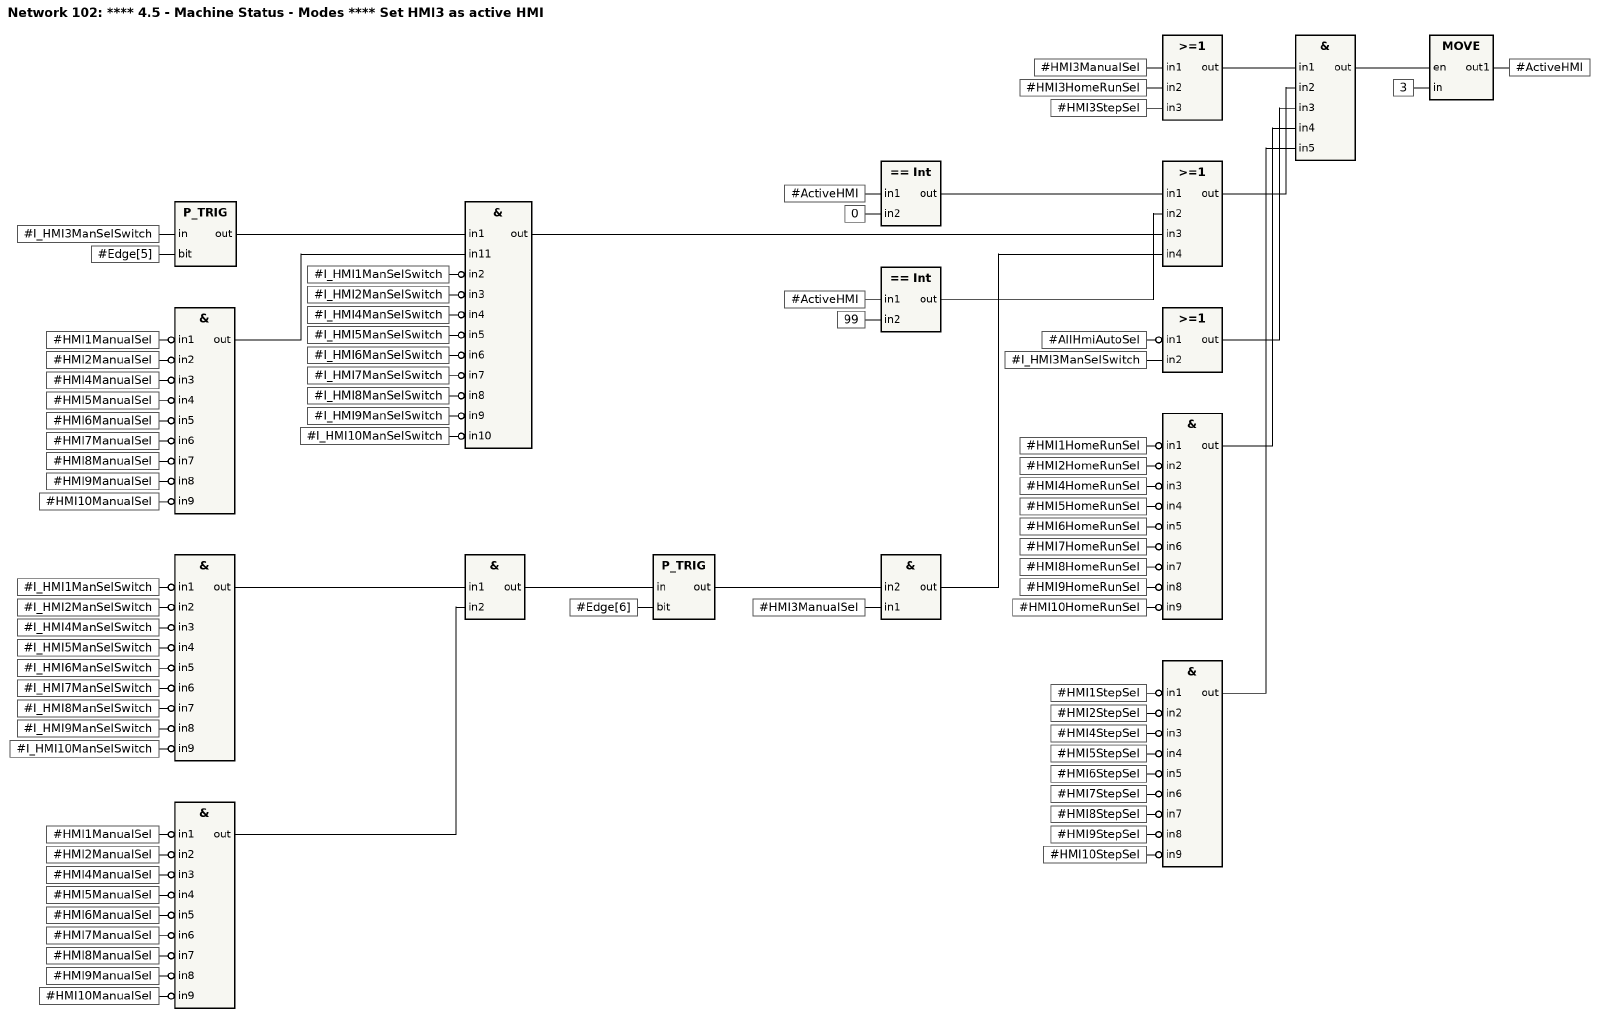
   #_w1 := #I_HMI3ManSelSwitch AND NOT #Edge[5];   // rising edge
   #Edge[5] := #I_HMI3ManSelSwitch;
   #_w2 := NOT #I_HMI1ManSelSwitch AND NOT #I_HMI2ManSelSwitch AND NOT #I_HMI4ManSelSwitch AND NOT #I_HMI5ManSelSwitch AND NOT #I_HMI6ManSelSwitch AND NOT #I_HMI7ManSelSwitch AND NOT #I_HMI8ManSelSwitch AND NOT #I_HMI9ManSelSwitch AND NOT #I_HMI10ManSelSwitch AND NOT #HMI1ManualSel AND NOT #HMI2ManualSel AND NOT #HMI4ManualSel AND NOT #HMI5ManualSel AND NOT #HMI6ManualSel AND NOT #HMI7ManualSel AND NOT #HMI8ManualSel AND NOT #HMI9ManualSel AND NOT #HMI10ManualSel;
   #_w3 := #_w2 AND NOT #Edge[6];   // rising edge
   #Edge[6] := #_w2;
   IF (#HMI3ManualSel OR #HMI3HomeRunSel OR #HMI3StepSel) AND ((#ActiveHMI = 0) OR (#ActiveHMI = 99) OR (#_w1 AND NOT #HMI1ManualSel AND NOT #HMI2ManualSel AND NOT #HMI4ManualSel AND NOT #HMI5ManualSel AND NOT #HMI6ManualSel AND NOT #HMI7ManualSel AND NOT #HMI8ManualSel AND NOT #HMI9ManualSel AND NOT #HMI10ManualSel AND NOT #I_HMI1ManSelSwitch AND NOT #I_HMI2ManSelSwitch AND NOT #I_HMI4ManSelSwitch AND NOT #I_HMI5ManSelSwitch AND NOT #I_HMI6ManSelSwitch AND NOT #I_HMI7ManSelSwitch AND NOT #I_HMI8ManSelSwitch AND NOT #I_HMI9ManSelSwitch AND NOT #I_HMI10ManSelSwitch) OR (#_w3 AND #HMI3ManualSel)) AND (NOT #AllHmiAutoSel OR #I_HMI3ManSelSwitch) AND NOT #HMI1HomeRunSel AND NOT #HMI2HomeRunSel AND NOT #HMI4HomeRunSel AND NOT #HMI5HomeRunSel AND NOT #HMI6HomeRunSel AND NOT #HMI7HomeRunSel AND NOT #HMI8HomeRunSel AND NOT #HMI9HomeRunSel AND NOT #HMI10HomeRunSel AND NOT #HMI1StepSel AND NOT #HMI2StepSel AND NOT #HMI4StepSel AND NOT #HMI5StepSel AND NOT #HMI6StepSel AND NOT #HMI7StepSel AND NOT #HMI8StepSel AND NOT #HMI9StepSel AND NOT #HMI10StepSel THEN
       #ActiveHMI := 3;
   END_IF;
END_REGION

REGION Network 103: **** 4.5 - Machine Status - Modes **** Set HMI4 as active HMI
   // Set HMI4 as active HMI
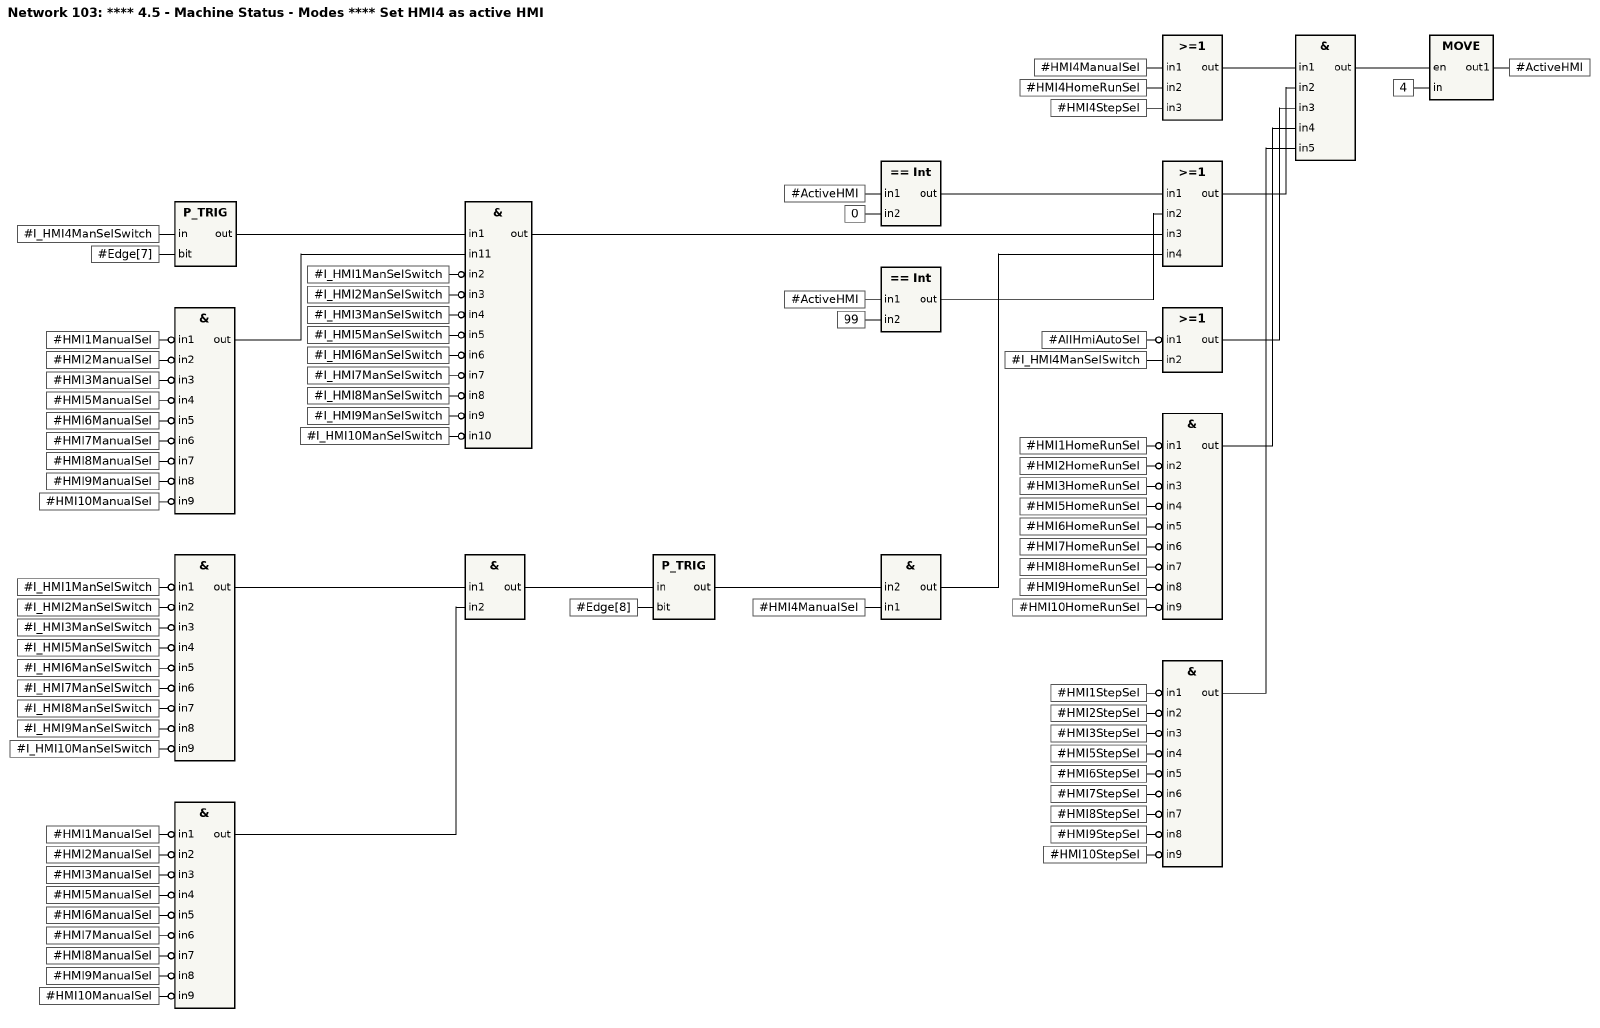
   #_w1 := #I_HMI4ManSelSwitch AND NOT #Edge[7];   // rising edge
   #Edge[7] := #I_HMI4ManSelSwitch;
   #_w2 := NOT #I_HMI1ManSelSwitch AND NOT #I_HMI2ManSelSwitch AND NOT #I_HMI3ManSelSwitch AND NOT #I_HMI5ManSelSwitch AND NOT #I_HMI6ManSelSwitch AND NOT #I_HMI7ManSelSwitch AND NOT #I_HMI8ManSelSwitch AND NOT #I_HMI9ManSelSwitch AND NOT #I_HMI10ManSelSwitch AND NOT #HMI1ManualSel AND NOT #HMI2ManualSel AND NOT #HMI3ManualSel AND NOT #HMI5ManualSel AND NOT #HMI6ManualSel AND NOT #HMI7ManualSel AND NOT #HMI8ManualSel AND NOT #HMI9ManualSel AND NOT #HMI10ManualSel;
   #_w3 := #_w2 AND NOT #Edge[8];   // rising edge
   #Edge[8] := #_w2;
   IF (#HMI4ManualSel OR #HMI4HomeRunSel OR #HMI4StepSel) AND ((#ActiveHMI = 0) OR (#ActiveHMI = 99) OR (#_w1 AND NOT #HMI1ManualSel AND NOT #HMI2ManualSel AND NOT #HMI3ManualSel AND NOT #HMI5ManualSel AND NOT #HMI6ManualSel AND NOT #HMI7ManualSel AND NOT #HMI8ManualSel AND NOT #HMI9ManualSel AND NOT #HMI10ManualSel AND NOT #I_HMI1ManSelSwitch AND NOT #I_HMI2ManSelSwitch AND NOT #I_HMI3ManSelSwitch AND NOT #I_HMI5ManSelSwitch AND NOT #I_HMI6ManSelSwitch AND NOT #I_HMI7ManSelSwitch AND NOT #I_HMI8ManSelSwitch AND NOT #I_HMI9ManSelSwitch AND NOT #I_HMI10ManSelSwitch) OR (#_w3 AND #HMI4ManualSel)) AND (NOT #AllHmiAutoSel OR #I_HMI4ManSelSwitch) AND NOT #HMI1HomeRunSel AND NOT #HMI2HomeRunSel AND NOT #HMI3HomeRunSel AND NOT #HMI5HomeRunSel AND NOT #HMI6HomeRunSel AND NOT #HMI7HomeRunSel AND NOT #HMI8HomeRunSel AND NOT #HMI9HomeRunSel AND NOT #HMI10HomeRunSel AND NOT #HMI1StepSel AND NOT #HMI2StepSel AND NOT #HMI3StepSel AND NOT #HMI5StepSel AND NOT #HMI6StepSel AND NOT #HMI7StepSel AND NOT #HMI8StepSel AND NOT #HMI9StepSel AND NOT #HMI10StepSel THEN
       #ActiveHMI := 4;
   END_IF;
END_REGION

REGION Network 104: **** 4.5 - Machine Status - Modes **** Set HMI5 as active HMI
   // Set HMI5 as active HMI
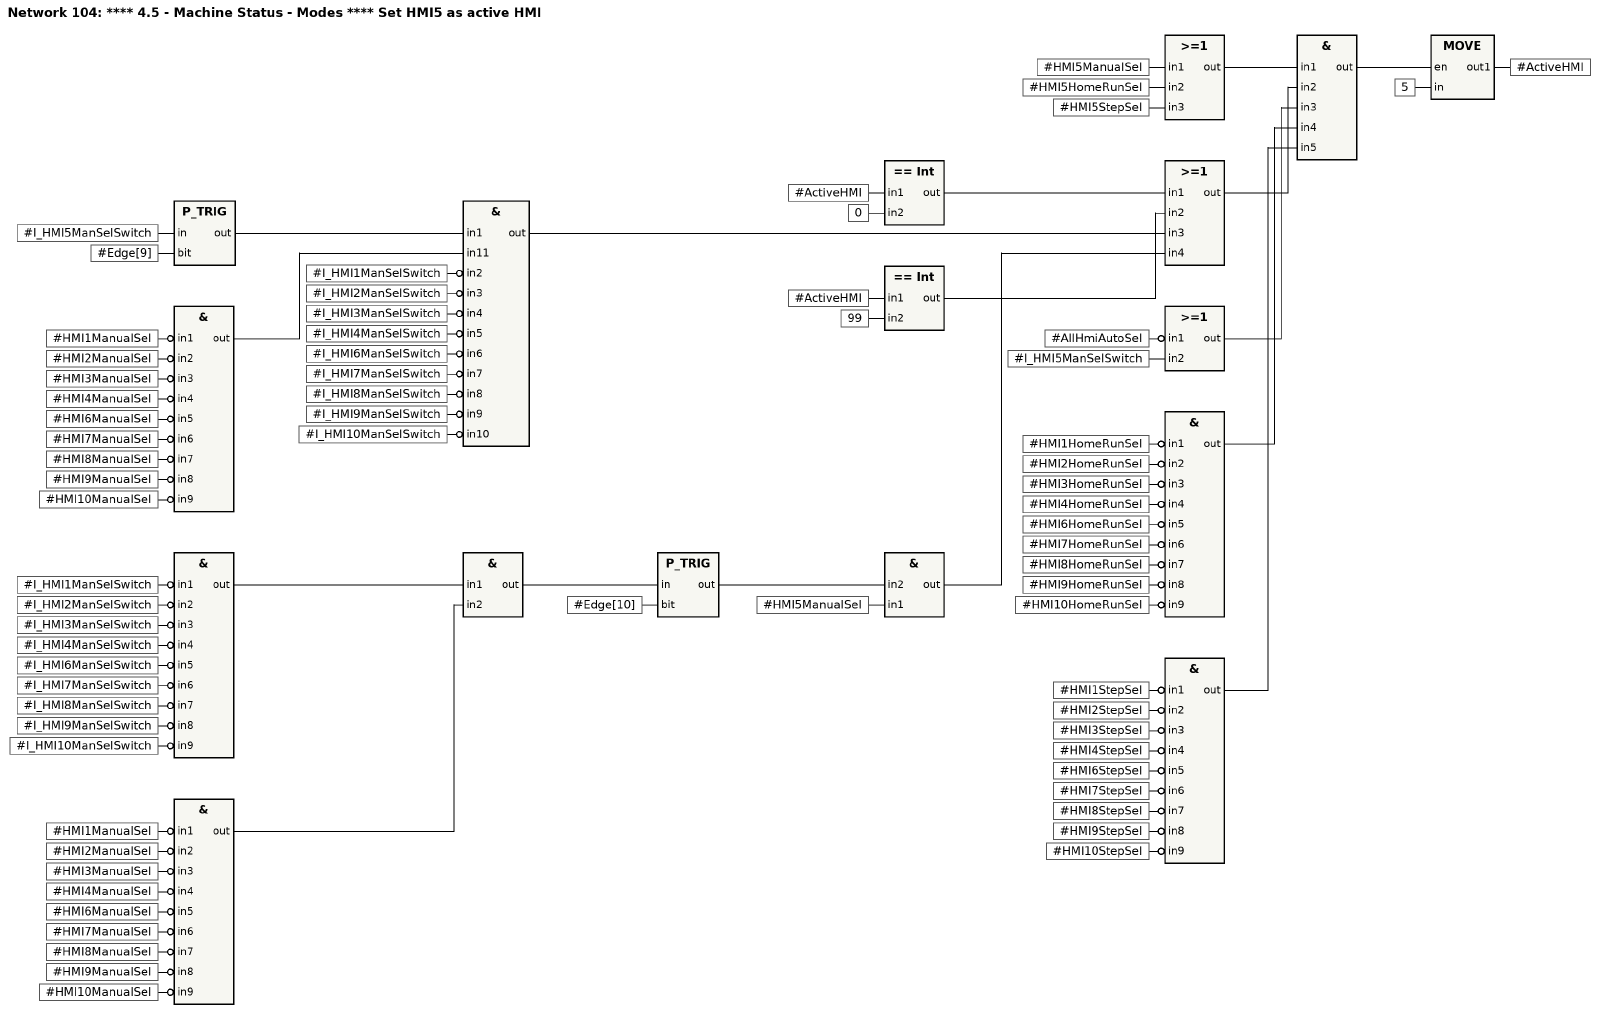
   #_w1 := #I_HMI5ManSelSwitch AND NOT #Edge[9];   // rising edge
   #Edge[9] := #I_HMI5ManSelSwitch;
   #_w2 := NOT #I_HMI1ManSelSwitch AND NOT #I_HMI2ManSelSwitch AND NOT #I_HMI3ManSelSwitch AND NOT #I_HMI4ManSelSwitch AND NOT #I_HMI6ManSelSwitch AND NOT #I_HMI7ManSelSwitch AND NOT #I_HMI8ManSelSwitch AND NOT #I_HMI9ManSelSwitch AND NOT #I_HMI10ManSelSwitch AND NOT #HMI1ManualSel AND NOT #HMI2ManualSel AND NOT #HMI3ManualSel AND NOT #HMI4ManualSel AND NOT #HMI6ManualSel AND NOT #HMI7ManualSel AND NOT #HMI8ManualSel AND NOT #HMI9ManualSel AND NOT #HMI10ManualSel;
   #_w3 := #_w2 AND NOT #Edge[10];   // rising edge
   #Edge[10] := #_w2;
   IF (#HMI5ManualSel OR #HMI5HomeRunSel OR #HMI5StepSel) AND ((#ActiveHMI = 0) OR (#ActiveHMI = 99) OR (#_w1 AND NOT #HMI1ManualSel AND NOT #HMI2ManualSel AND NOT #HMI3ManualSel AND NOT #HMI4ManualSel AND NOT #HMI6ManualSel AND NOT #HMI7ManualSel AND NOT #HMI8ManualSel AND NOT #HMI9ManualSel AND NOT #HMI10ManualSel AND NOT #I_HMI1ManSelSwitch AND NOT #I_HMI2ManSelSwitch AND NOT #I_HMI3ManSelSwitch AND NOT #I_HMI4ManSelSwitch AND NOT #I_HMI6ManSelSwitch AND NOT #I_HMI7ManSelSwitch AND NOT #I_HMI8ManSelSwitch AND NOT #I_HMI9ManSelSwitch AND NOT #I_HMI10ManSelSwitch) OR (#_w3 AND #HMI5ManualSel)) AND (NOT #AllHmiAutoSel OR #I_HMI5ManSelSwitch) AND NOT #HMI1HomeRunSel AND NOT #HMI2HomeRunSel AND NOT #HMI3HomeRunSel AND NOT #HMI4HomeRunSel AND NOT #HMI6HomeRunSel AND NOT #HMI7HomeRunSel AND NOT #HMI8HomeRunSel AND NOT #HMI9HomeRunSel AND NOT #HMI10HomeRunSel AND NOT #HMI1StepSel AND NOT #HMI2StepSel AND NOT #HMI3StepSel AND NOT #HMI4StepSel AND NOT #HMI6StepSel AND NOT #HMI7StepSel AND NOT #HMI8StepSel AND NOT #HMI9StepSel AND NOT #HMI10StepSel THEN
       #ActiveHMI := 5;
   END_IF;
END_REGION

REGION Network 105: **** 4.5 - Machine Status - Modes **** Set HMI6 as active HMI
   // Set HMI6 as active HMI
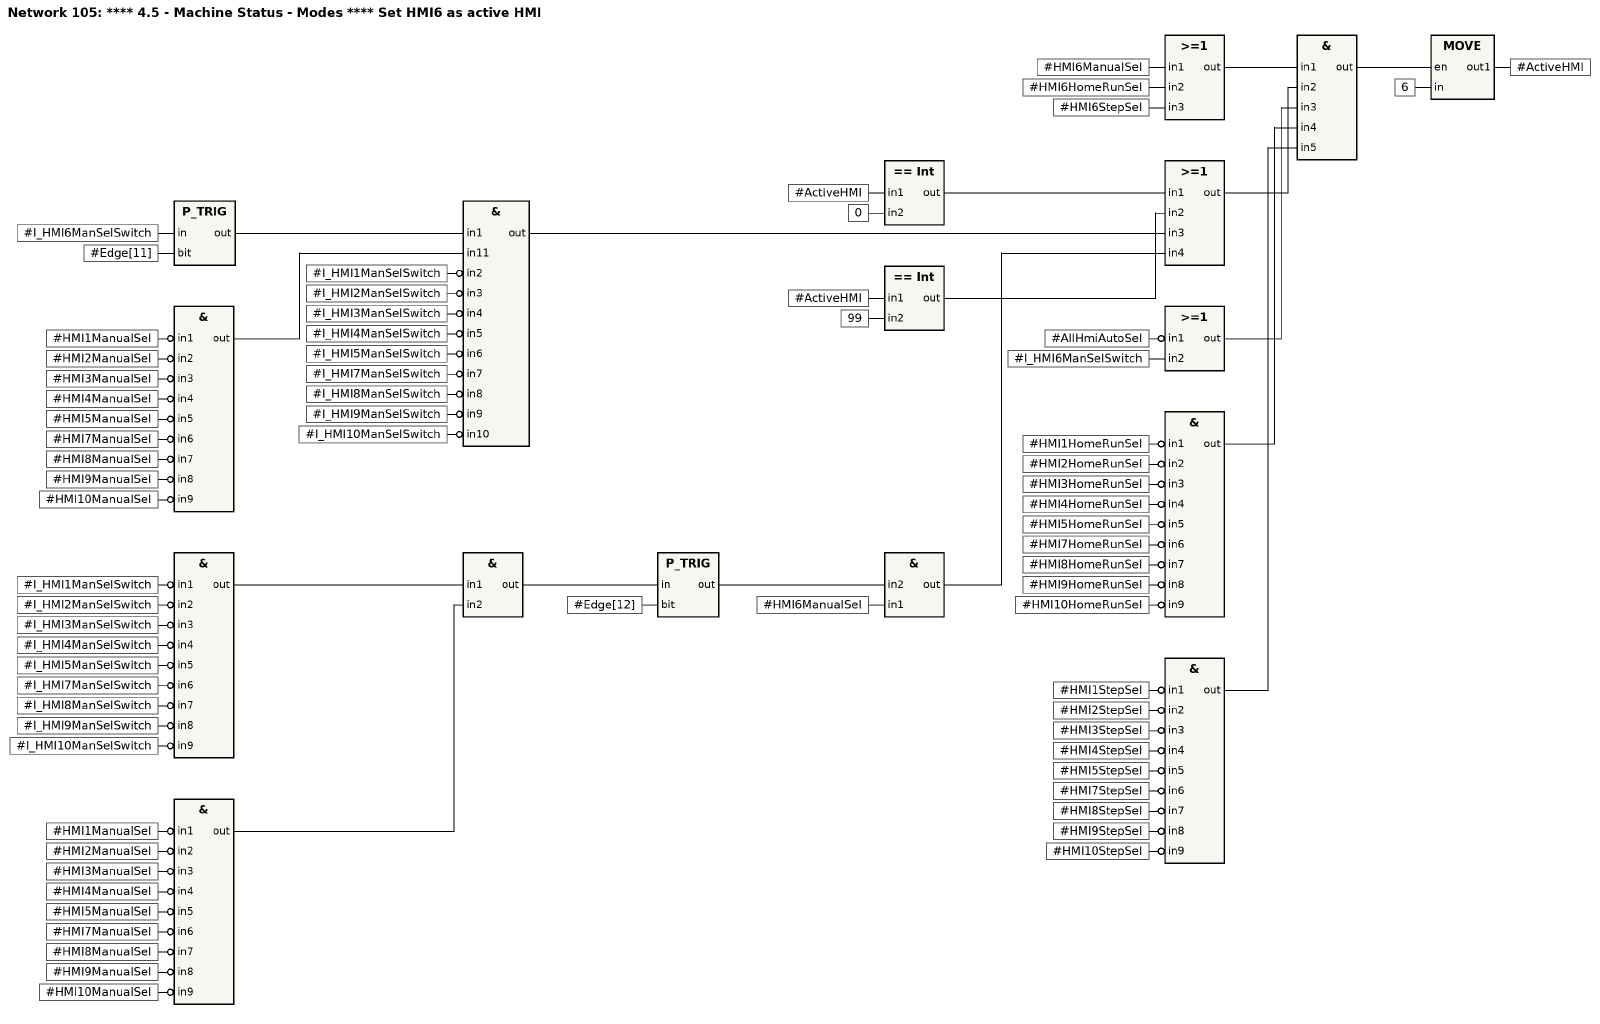
   #_w1 := #I_HMI6ManSelSwitch AND NOT #Edge[11];   // rising edge
   #Edge[11] := #I_HMI6ManSelSwitch;
   #_w2 := NOT #I_HMI1ManSelSwitch AND NOT #I_HMI2ManSelSwitch AND NOT #I_HMI3ManSelSwitch AND NOT #I_HMI4ManSelSwitch AND NOT #I_HMI5ManSelSwitch AND NOT #I_HMI7ManSelSwitch AND NOT #I_HMI8ManSelSwitch AND NOT #I_HMI9ManSelSwitch AND NOT #I_HMI10ManSelSwitch AND NOT #HMI1ManualSel AND NOT #HMI2ManualSel AND NOT #HMI3ManualSel AND NOT #HMI4ManualSel AND NOT #HMI5ManualSel AND NOT #HMI7ManualSel AND NOT #HMI8ManualSel AND NOT #HMI9ManualSel AND NOT #HMI10ManualSel;
   #_w3 := #_w2 AND NOT #Edge[12];   // rising edge
   #Edge[12] := #_w2;
   IF (#HMI6ManualSel OR #HMI6HomeRunSel OR #HMI6StepSel) AND ((#ActiveHMI = 0) OR (#ActiveHMI = 99) OR (#_w1 AND NOT #HMI1ManualSel AND NOT #HMI2ManualSel AND NOT #HMI3ManualSel AND NOT #HMI4ManualSel AND NOT #HMI5ManualSel AND NOT #HMI7ManualSel AND NOT #HMI8ManualSel AND NOT #HMI9ManualSel AND NOT #HMI10ManualSel AND NOT #I_HMI1ManSelSwitch AND NOT #I_HMI2ManSelSwitch AND NOT #I_HMI3ManSelSwitch AND NOT #I_HMI4ManSelSwitch AND NOT #I_HMI5ManSelSwitch AND NOT #I_HMI7ManSelSwitch AND NOT #I_HMI8ManSelSwitch AND NOT #I_HMI9ManSelSwitch AND NOT #I_HMI10ManSelSwitch) OR (#_w3 AND #HMI6ManualSel)) AND (NOT #AllHmiAutoSel OR #I_HMI6ManSelSwitch) AND NOT #HMI1HomeRunSel AND NOT #HMI2HomeRunSel AND NOT #HMI3HomeRunSel AND NOT #HMI4HomeRunSel AND NOT #HMI5HomeRunSel AND NOT #HMI7HomeRunSel AND NOT #HMI8HomeRunSel AND NOT #HMI9HomeRunSel AND NOT #HMI10HomeRunSel AND NOT #HMI1StepSel AND NOT #HMI2StepSel AND NOT #HMI3StepSel AND NOT #HMI4StepSel AND NOT #HMI5StepSel AND NOT #HMI7StepSel AND NOT #HMI8StepSel AND NOT #HMI9StepSel AND NOT #HMI10StepSel THEN
       #ActiveHMI := 6;
   END_IF;
END_REGION

REGION Network 106: **** 4.5 - Machine Status - Modes **** Set HMI7 as active HMI
   // Set HMI7 as active HMI
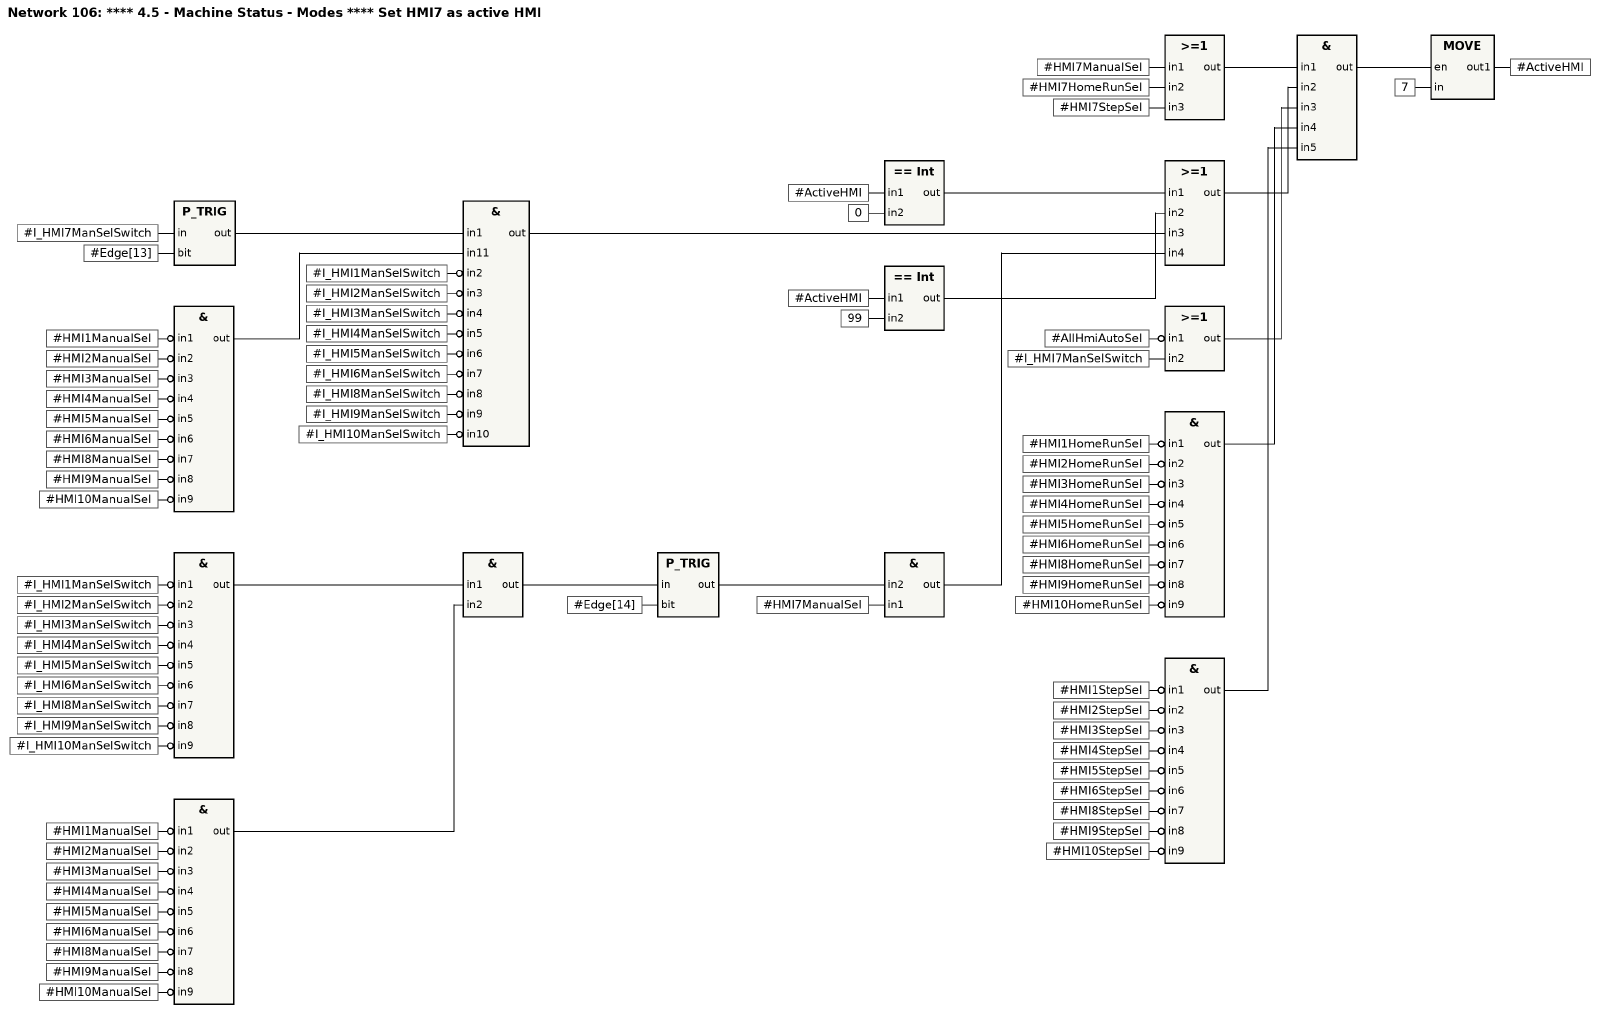
   #_w1 := #I_HMI7ManSelSwitch AND NOT #Edge[13];   // rising edge
   #Edge[13] := #I_HMI7ManSelSwitch;
   #_w2 := NOT #I_HMI1ManSelSwitch AND NOT #I_HMI2ManSelSwitch AND NOT #I_HMI3ManSelSwitch AND NOT #I_HMI4ManSelSwitch AND NOT #I_HMI5ManSelSwitch AND NOT #I_HMI6ManSelSwitch AND NOT #I_HMI8ManSelSwitch AND NOT #I_HMI9ManSelSwitch AND NOT #I_HMI10ManSelSwitch AND NOT #HMI1ManualSel AND NOT #HMI2ManualSel AND NOT #HMI3ManualSel AND NOT #HMI4ManualSel AND NOT #HMI5ManualSel AND NOT #HMI6ManualSel AND NOT #HMI8ManualSel AND NOT #HMI9ManualSel AND NOT #HMI10ManualSel;
   #_w3 := #_w2 AND NOT #Edge[14];   // rising edge
   #Edge[14] := #_w2;
   IF (#HMI7ManualSel OR #HMI7HomeRunSel OR #HMI7StepSel) AND ((#ActiveHMI = 0) OR (#ActiveHMI = 99) OR (#_w1 AND NOT #HMI1ManualSel AND NOT #HMI2ManualSel AND NOT #HMI3ManualSel AND NOT #HMI4ManualSel AND NOT #HMI5ManualSel AND NOT #HMI6ManualSel AND NOT #HMI8ManualSel AND NOT #HMI9ManualSel AND NOT #HMI10ManualSel AND NOT #I_HMI1ManSelSwitch AND NOT #I_HMI2ManSelSwitch AND NOT #I_HMI3ManSelSwitch AND NOT #I_HMI4ManSelSwitch AND NOT #I_HMI5ManSelSwitch AND NOT #I_HMI6ManSelSwitch AND NOT #I_HMI8ManSelSwitch AND NOT #I_HMI9ManSelSwitch AND NOT #I_HMI10ManSelSwitch) OR (#_w3 AND #HMI7ManualSel)) AND (NOT #AllHmiAutoSel OR #I_HMI7ManSelSwitch) AND NOT #HMI1HomeRunSel AND NOT #HMI2HomeRunSel AND NOT #HMI3HomeRunSel AND NOT #HMI4HomeRunSel AND NOT #HMI5HomeRunSel AND NOT #HMI6HomeRunSel AND NOT #HMI8HomeRunSel AND NOT #HMI9HomeRunSel AND NOT #HMI10HomeRunSel AND NOT #HMI1StepSel AND NOT #HMI2StepSel AND NOT #HMI3StepSel AND NOT #HMI4StepSel AND NOT #HMI5StepSel AND NOT #HMI6StepSel AND NOT #HMI8StepSel AND NOT #HMI9StepSel AND NOT #HMI10StepSel THEN
       #ActiveHMI := 7;
   END_IF;
END_REGION

REGION Network 107: **** 4.5 - Machine Status - Modes **** Set HMI8 as active HMI
   // Set HMI8 as active HMI
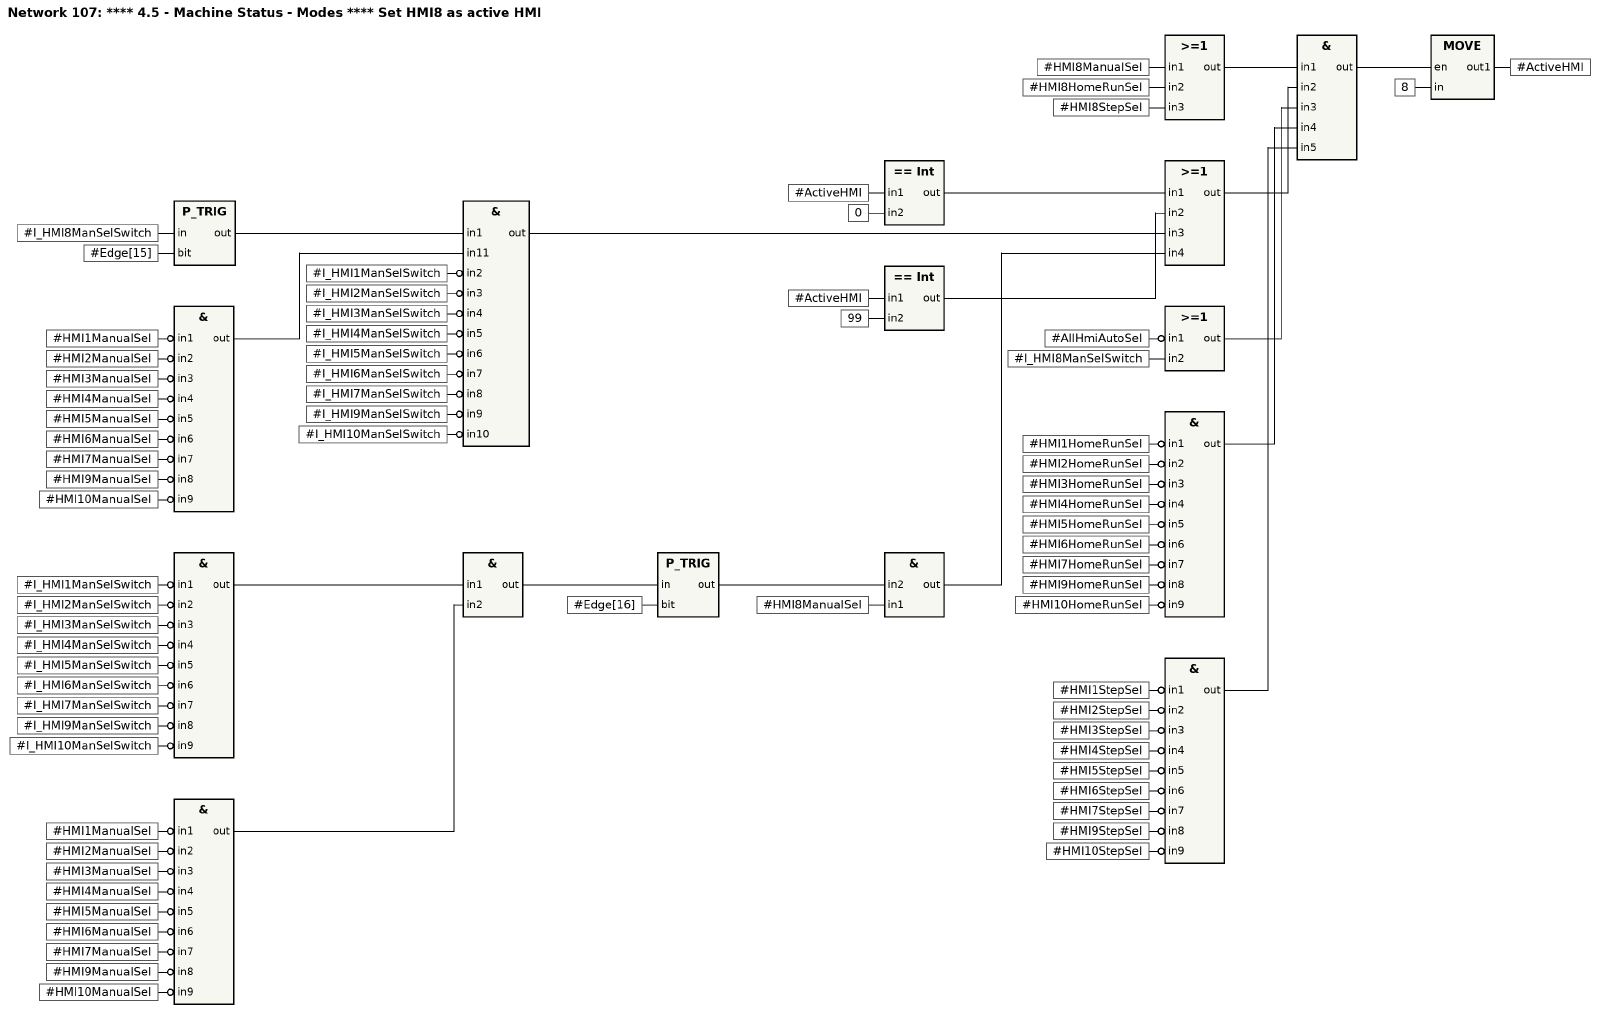
   #_w1 := #I_HMI8ManSelSwitch AND NOT #Edge[15];   // rising edge
   #Edge[15] := #I_HMI8ManSelSwitch;
   #_w2 := NOT #I_HMI1ManSelSwitch AND NOT #I_HMI2ManSelSwitch AND NOT #I_HMI3ManSelSwitch AND NOT #I_HMI4ManSelSwitch AND NOT #I_HMI5ManSelSwitch AND NOT #I_HMI6ManSelSwitch AND NOT #I_HMI7ManSelSwitch AND NOT #I_HMI9ManSelSwitch AND NOT #I_HMI10ManSelSwitch AND NOT #HMI1ManualSel AND NOT #HMI2ManualSel AND NOT #HMI3ManualSel AND NOT #HMI4ManualSel AND NOT #HMI5ManualSel AND NOT #HMI6ManualSel AND NOT #HMI7ManualSel AND NOT #HMI9ManualSel AND NOT #HMI10ManualSel;
   #_w3 := #_w2 AND NOT #Edge[16];   // rising edge
   #Edge[16] := #_w2;
   IF (#HMI8ManualSel OR #HMI8HomeRunSel OR #HMI8StepSel) AND ((#ActiveHMI = 0) OR (#ActiveHMI = 99) OR (#_w1 AND NOT #HMI1ManualSel AND NOT #HMI2ManualSel AND NOT #HMI3ManualSel AND NOT #HMI4ManualSel AND NOT #HMI5ManualSel AND NOT #HMI6ManualSel AND NOT #HMI7ManualSel AND NOT #HMI9ManualSel AND NOT #HMI10ManualSel AND NOT #I_HMI1ManSelSwitch AND NOT #I_HMI2ManSelSwitch AND NOT #I_HMI3ManSelSwitch AND NOT #I_HMI4ManSelSwitch AND NOT #I_HMI5ManSelSwitch AND NOT #I_HMI6ManSelSwitch AND NOT #I_HMI7ManSelSwitch AND NOT #I_HMI9ManSelSwitch AND NOT #I_HMI10ManSelSwitch) OR (#_w3 AND #HMI8ManualSel)) AND (NOT #AllHmiAutoSel OR #I_HMI8ManSelSwitch) AND NOT #HMI1HomeRunSel AND NOT #HMI2HomeRunSel AND NOT #HMI3HomeRunSel AND NOT #HMI4HomeRunSel AND NOT #HMI5HomeRunSel AND NOT #HMI6HomeRunSel AND NOT #HMI7HomeRunSel AND NOT #HMI9HomeRunSel AND NOT #HMI10HomeRunSel AND NOT #HMI1StepSel AND NOT #HMI2StepSel AND NOT #HMI3StepSel AND NOT #HMI4StepSel AND NOT #HMI5StepSel AND NOT #HMI6StepSel AND NOT #HMI7StepSel AND NOT #HMI9StepSel AND NOT #HMI10StepSel THEN
       #ActiveHMI := 8;
   END_IF;
END_REGION

REGION Network 108: **** 4.5 - Machine Status - Modes **** Set HMI9 as active HMI
   // Set HMI9 as active HMI
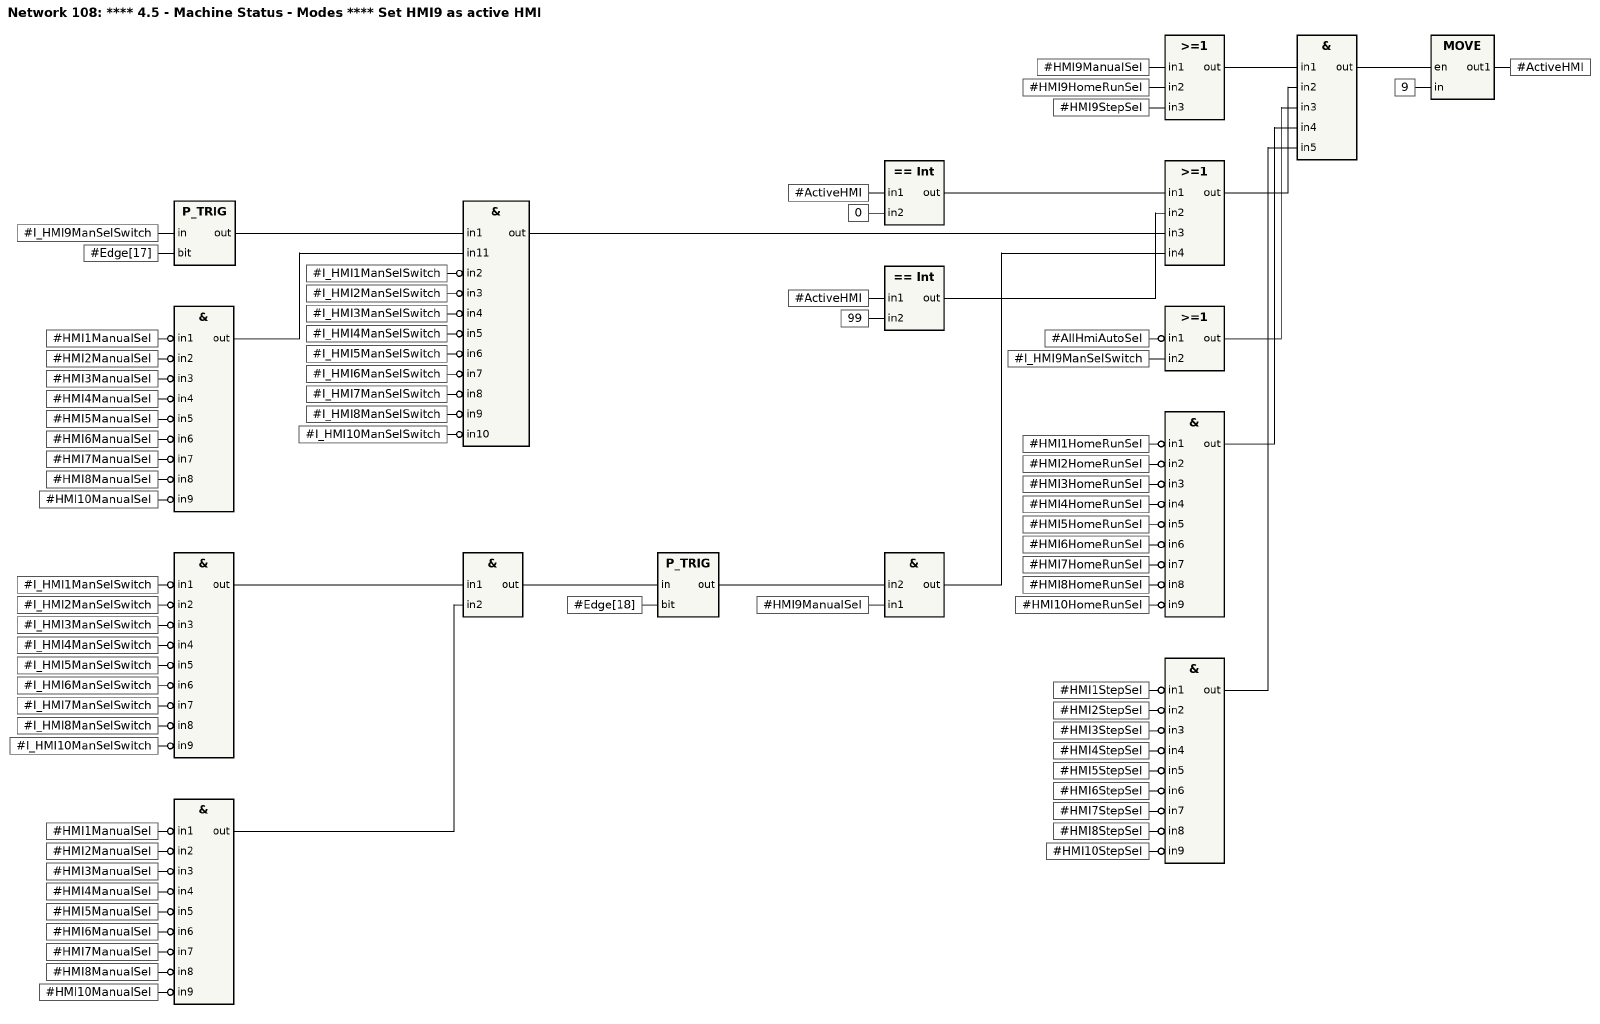
   #_w1 := #I_HMI9ManSelSwitch AND NOT #Edge[17];   // rising edge
   #Edge[17] := #I_HMI9ManSelSwitch;
   #_w2 := NOT #I_HMI1ManSelSwitch AND NOT #I_HMI2ManSelSwitch AND NOT #I_HMI3ManSelSwitch AND NOT #I_HMI4ManSelSwitch AND NOT #I_HMI5ManSelSwitch AND NOT #I_HMI6ManSelSwitch AND NOT #I_HMI7ManSelSwitch AND NOT #I_HMI8ManSelSwitch AND NOT #I_HMI10ManSelSwitch AND NOT #HMI1ManualSel AND NOT #HMI2ManualSel AND NOT #HMI3ManualSel AND NOT #HMI4ManualSel AND NOT #HMI5ManualSel AND NOT #HMI6ManualSel AND NOT #HMI7ManualSel AND NOT #HMI8ManualSel AND NOT #HMI10ManualSel;
   #_w3 := #_w2 AND NOT #Edge[18];   // rising edge
   #Edge[18] := #_w2;
   IF (#HMI9ManualSel OR #HMI9HomeRunSel OR #HMI9StepSel) AND ((#ActiveHMI = 0) OR (#ActiveHMI = 99) OR (#_w1 AND NOT #HMI1ManualSel AND NOT #HMI2ManualSel AND NOT #HMI3ManualSel AND NOT #HMI4ManualSel AND NOT #HMI5ManualSel AND NOT #HMI6ManualSel AND NOT #HMI7ManualSel AND NOT #HMI8ManualSel AND NOT #HMI10ManualSel AND NOT #I_HMI1ManSelSwitch AND NOT #I_HMI2ManSelSwitch AND NOT #I_HMI3ManSelSwitch AND NOT #I_HMI4ManSelSwitch AND NOT #I_HMI5ManSelSwitch AND NOT #I_HMI6ManSelSwitch AND NOT #I_HMI7ManSelSwitch AND NOT #I_HMI8ManSelSwitch AND NOT #I_HMI10ManSelSwitch) OR (#_w3 AND #HMI9ManualSel)) AND (NOT #AllHmiAutoSel OR #I_HMI9ManSelSwitch) AND NOT #HMI1HomeRunSel AND NOT #HMI2HomeRunSel AND NOT #HMI3HomeRunSel AND NOT #HMI4HomeRunSel AND NOT #HMI5HomeRunSel AND NOT #HMI6HomeRunSel AND NOT #HMI7HomeRunSel AND NOT #HMI8HomeRunSel AND NOT #HMI10HomeRunSel AND NOT #HMI1StepSel AND NOT #HMI2StepSel AND NOT #HMI3StepSel AND NOT #HMI4StepSel AND NOT #HMI5StepSel AND NOT #HMI6StepSel AND NOT #HMI7StepSel AND NOT #HMI8StepSel AND NOT #HMI10StepSel THEN
       #ActiveHMI := 9;
   END_IF;
END_REGION

REGION Network 109: **** 4.5 - Machine Status - Modes **** Set HMI10 as active HMI
   // Set HMI10 as active HMI
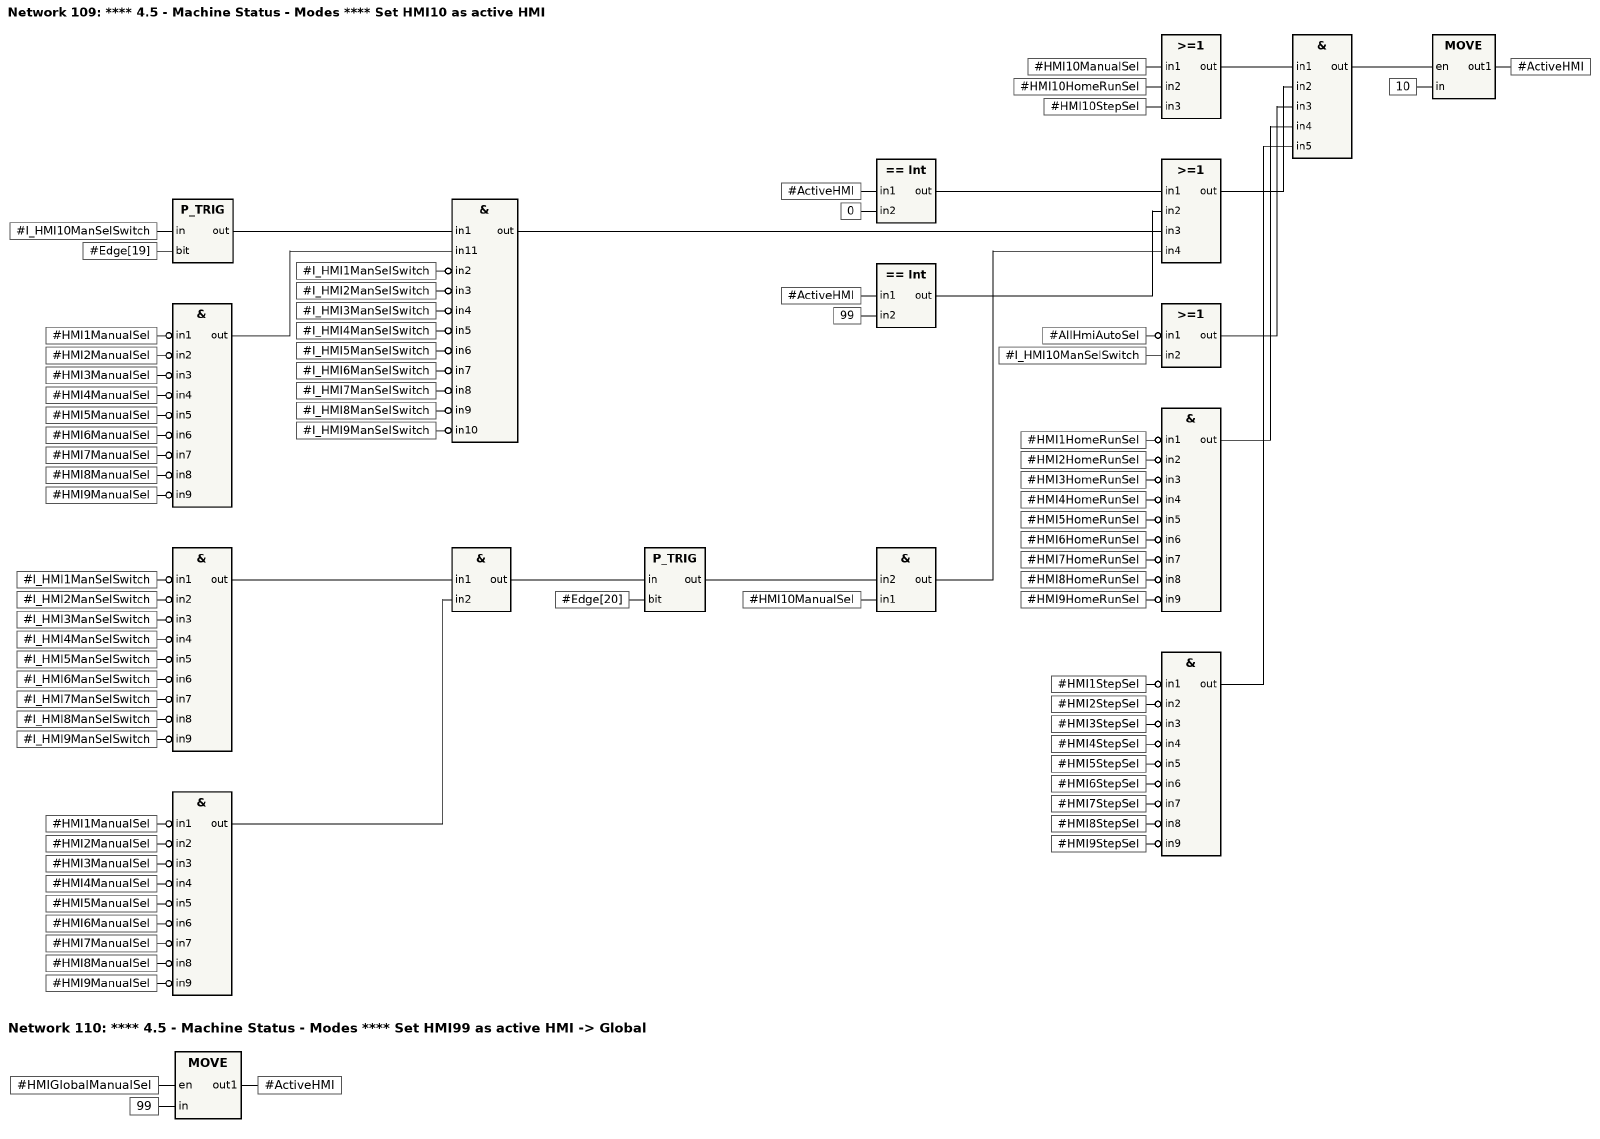
   #_w1 := #I_HMI10ManSelSwitch AND NOT #Edge[19];   // rising edge
   #Edge[19] := #I_HMI10ManSelSwitch;
   #_w2 := NOT #I_HMI1ManSelSwitch AND NOT #I_HMI2ManSelSwitch AND NOT #I_HMI3ManSelSwitch AND NOT #I_HMI4ManSelSwitch AND NOT #I_HMI5ManSelSwitch AND NOT #I_HMI6ManSelSwitch AND NOT #I_HMI7ManSelSwitch AND NOT #I_HMI8ManSelSwitch AND NOT #I_HMI9ManSelSwitch AND NOT #HMI1ManualSel AND NOT #HMI2ManualSel AND NOT #HMI3ManualSel AND NOT #HMI4ManualSel AND NOT #HMI5ManualSel AND NOT #HMI6ManualSel AND NOT #HMI7ManualSel AND NOT #HMI8ManualSel AND NOT #HMI9ManualSel;
   #_w3 := #_w2 AND NOT #Edge[20];   // rising edge
   #Edge[20] := #_w2;
   IF (#HMI10ManualSel OR #HMI10HomeRunSel OR #HMI10StepSel) AND ((#ActiveHMI = 0) OR (#ActiveHMI = 99) OR (#_w1 AND NOT #HMI1ManualSel AND NOT #HMI2ManualSel AND NOT #HMI3ManualSel AND NOT #HMI4ManualSel AND NOT #HMI5ManualSel AND NOT #HMI6ManualSel AND NOT #HMI7ManualSel AND NOT #HMI8ManualSel AND NOT #HMI9ManualSel AND NOT #I_HMI1ManSelSwitch AND NOT #I_HMI2ManSelSwitch AND NOT #I_HMI3ManSelSwitch AND NOT #I_HMI4ManSelSwitch AND NOT #I_HMI5ManSelSwitch AND NOT #I_HMI6ManSelSwitch AND NOT #I_HMI7ManSelSwitch AND NOT #I_HMI8ManSelSwitch AND NOT #I_HMI9ManSelSwitch) OR (#_w3 AND #HMI10ManualSel)) AND (NOT #AllHmiAutoSel OR #I_HMI10ManSelSwitch) AND NOT #HMI1HomeRunSel AND NOT #HMI2HomeRunSel AND NOT #HMI3HomeRunSel AND NOT #HMI4HomeRunSel AND NOT #HMI5HomeRunSel AND NOT #HMI6HomeRunSel AND NOT #HMI7HomeRunSel AND NOT #HMI8HomeRunSel AND NOT #HMI9HomeRunSel AND NOT #HMI1StepSel AND NOT #HMI2StepSel AND NOT #HMI3StepSel AND NOT #HMI4StepSel AND NOT #HMI5StepSel AND NOT #HMI6StepSel AND NOT #HMI7StepSel AND NOT #HMI8StepSel AND NOT #HMI9StepSel THEN
       #ActiveHMI := 10;
   END_IF;
END_REGION

REGION Network 110: **** 4.5 - Machine Status - Modes **** Set HMI99 as active HMI -> Global
   IF #HMIGlobalManualSel THEN #ActiveHMI := 99; END_IF;
END_REGION

REGION Network 111: **** 4.5 - Machine Status - Modes **** Set Manual selected if one of the HMI is active
   // Set Manual selected if one of the HMI is active
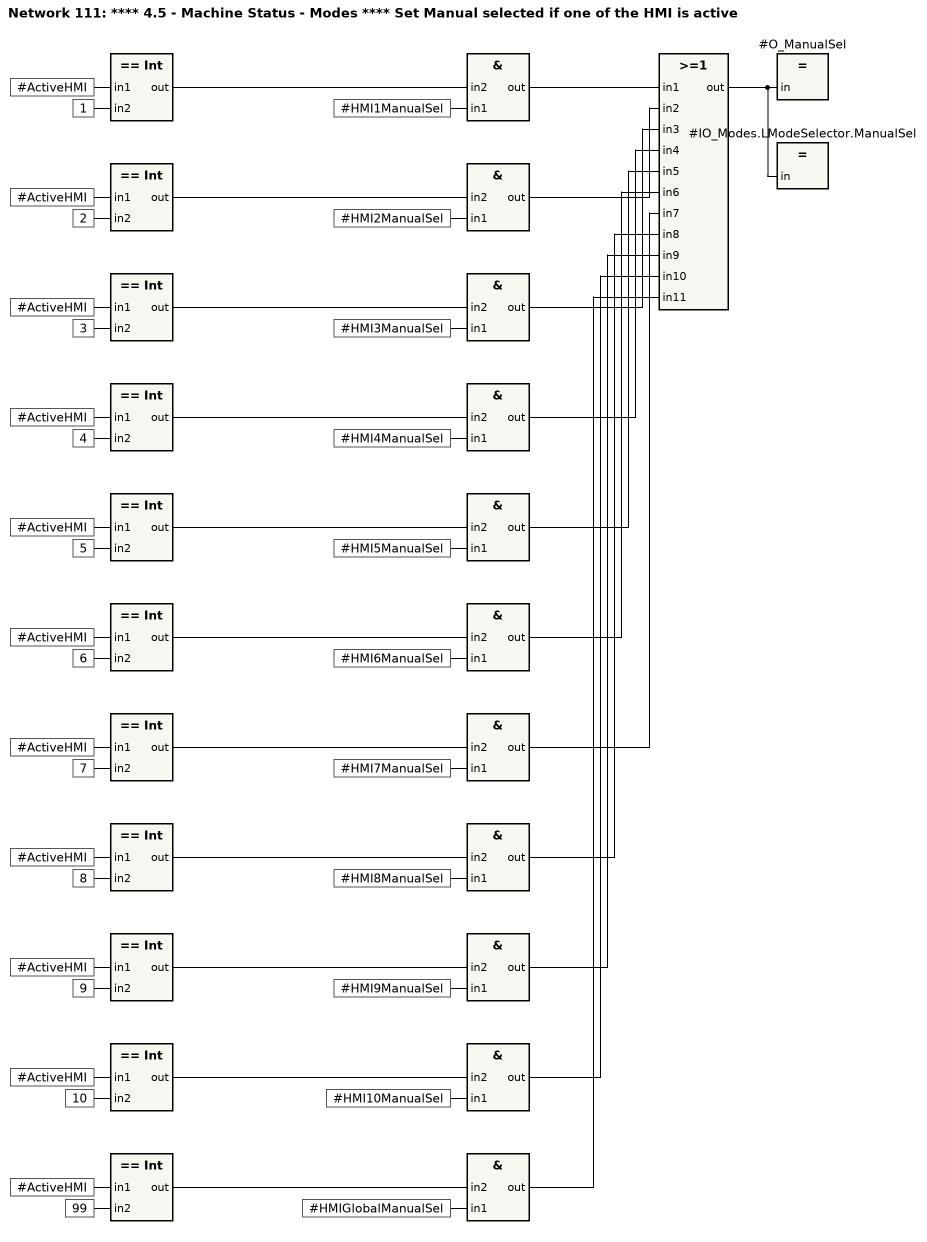
   #O_ManualSel := ((#ActiveHMI = 1) AND #HMI1ManualSel) OR ((#ActiveHMI = 2) AND #HMI2ManualSel) OR ((#ActiveHMI = 3) AND #HMI3ManualSel) OR ((#ActiveHMI = 4) AND #HMI4ManualSel) OR ((#ActiveHMI = 5) AND #HMI5ManualSel) OR ((#ActiveHMI = 6) AND #HMI6ManualSel) OR ((#ActiveHMI = 7) AND #HMI7ManualSel) OR ((#ActiveHMI = 8) AND #HMI8ManualSel) OR ((#ActiveHMI = 9) AND #HMI9ManualSel) OR ((#ActiveHMI = 10) AND #HMI10ManualSel) OR ((#ActiveHMI = 99) AND #HMIGlobalManualSel);
   #IO_Modes.LModeSelector.ManualSel := #O_ManualSel;
END_REGION

REGION Network 112: **** 4.6 - Machine Status - Indications **** Animation
   // Animation
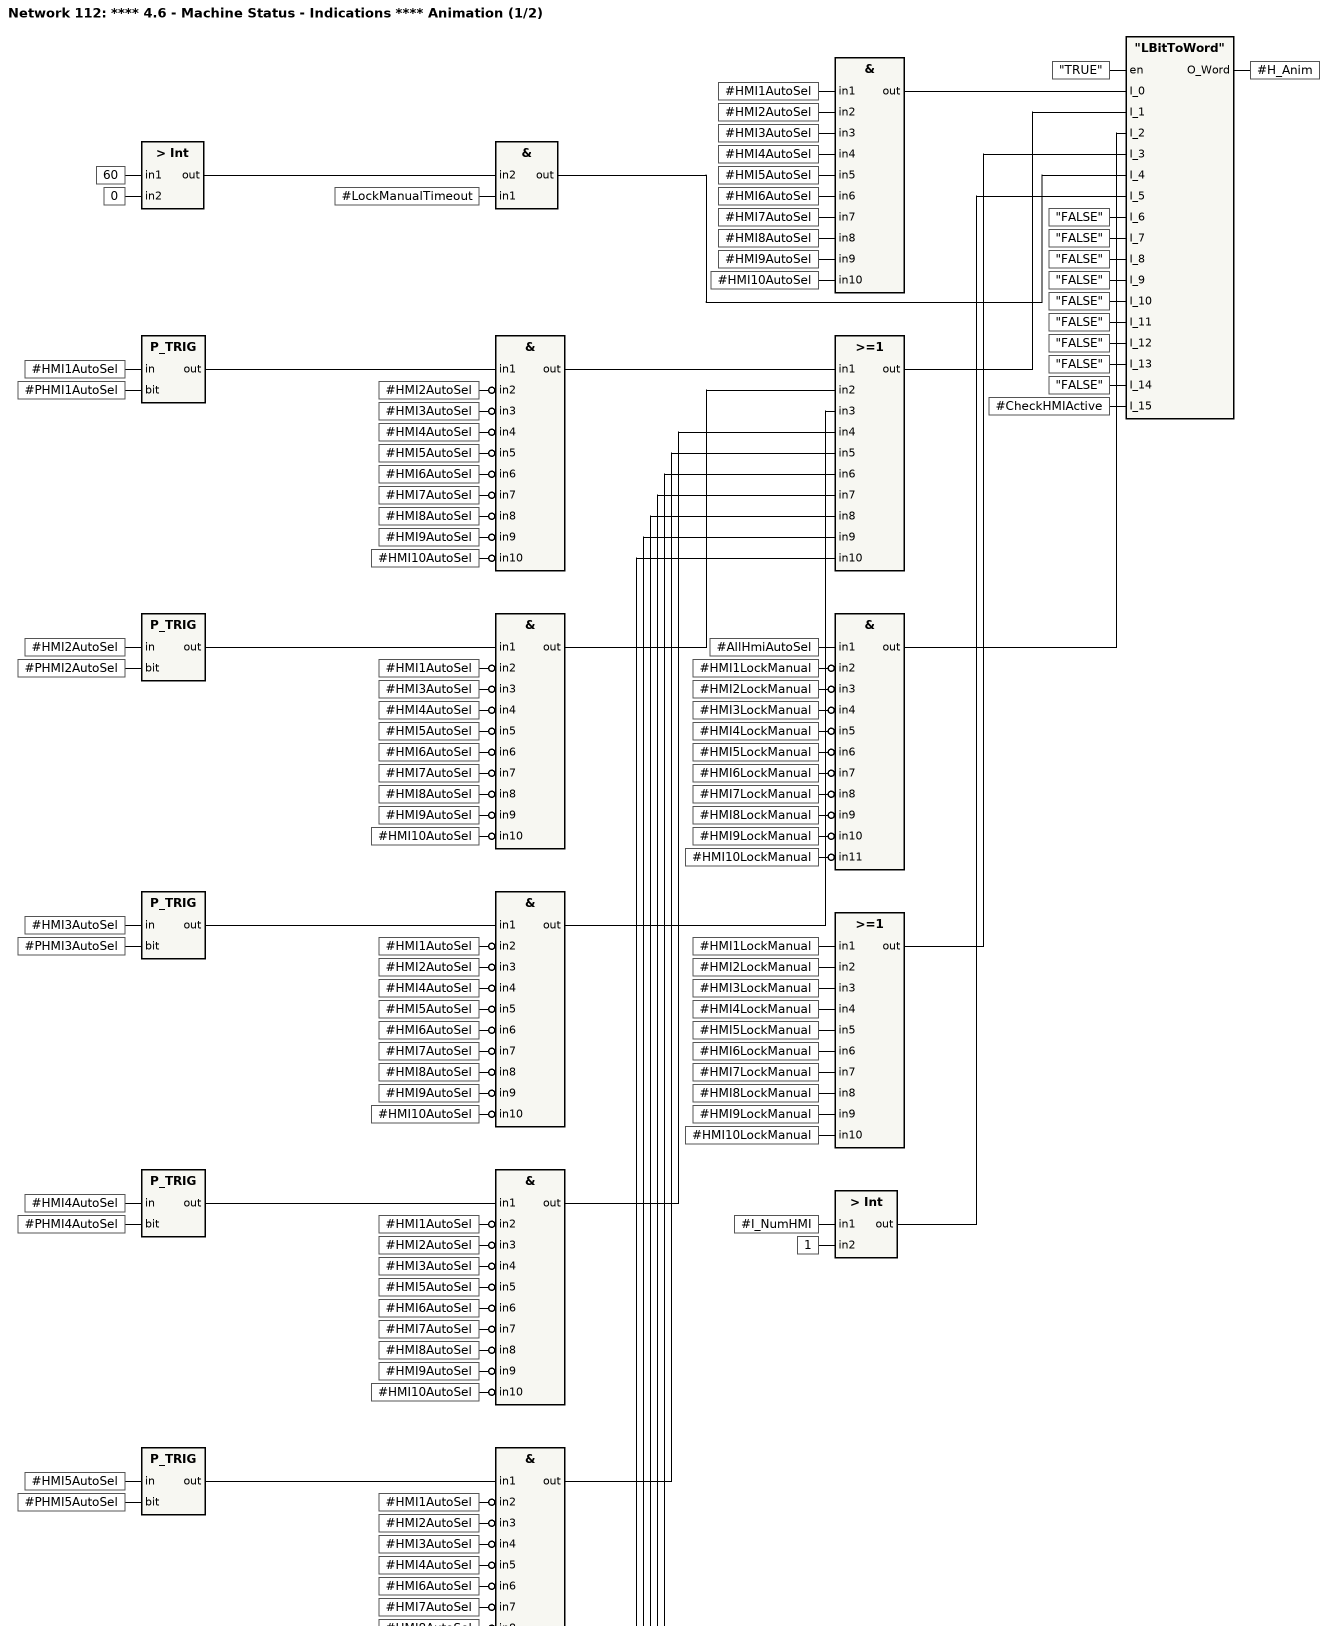
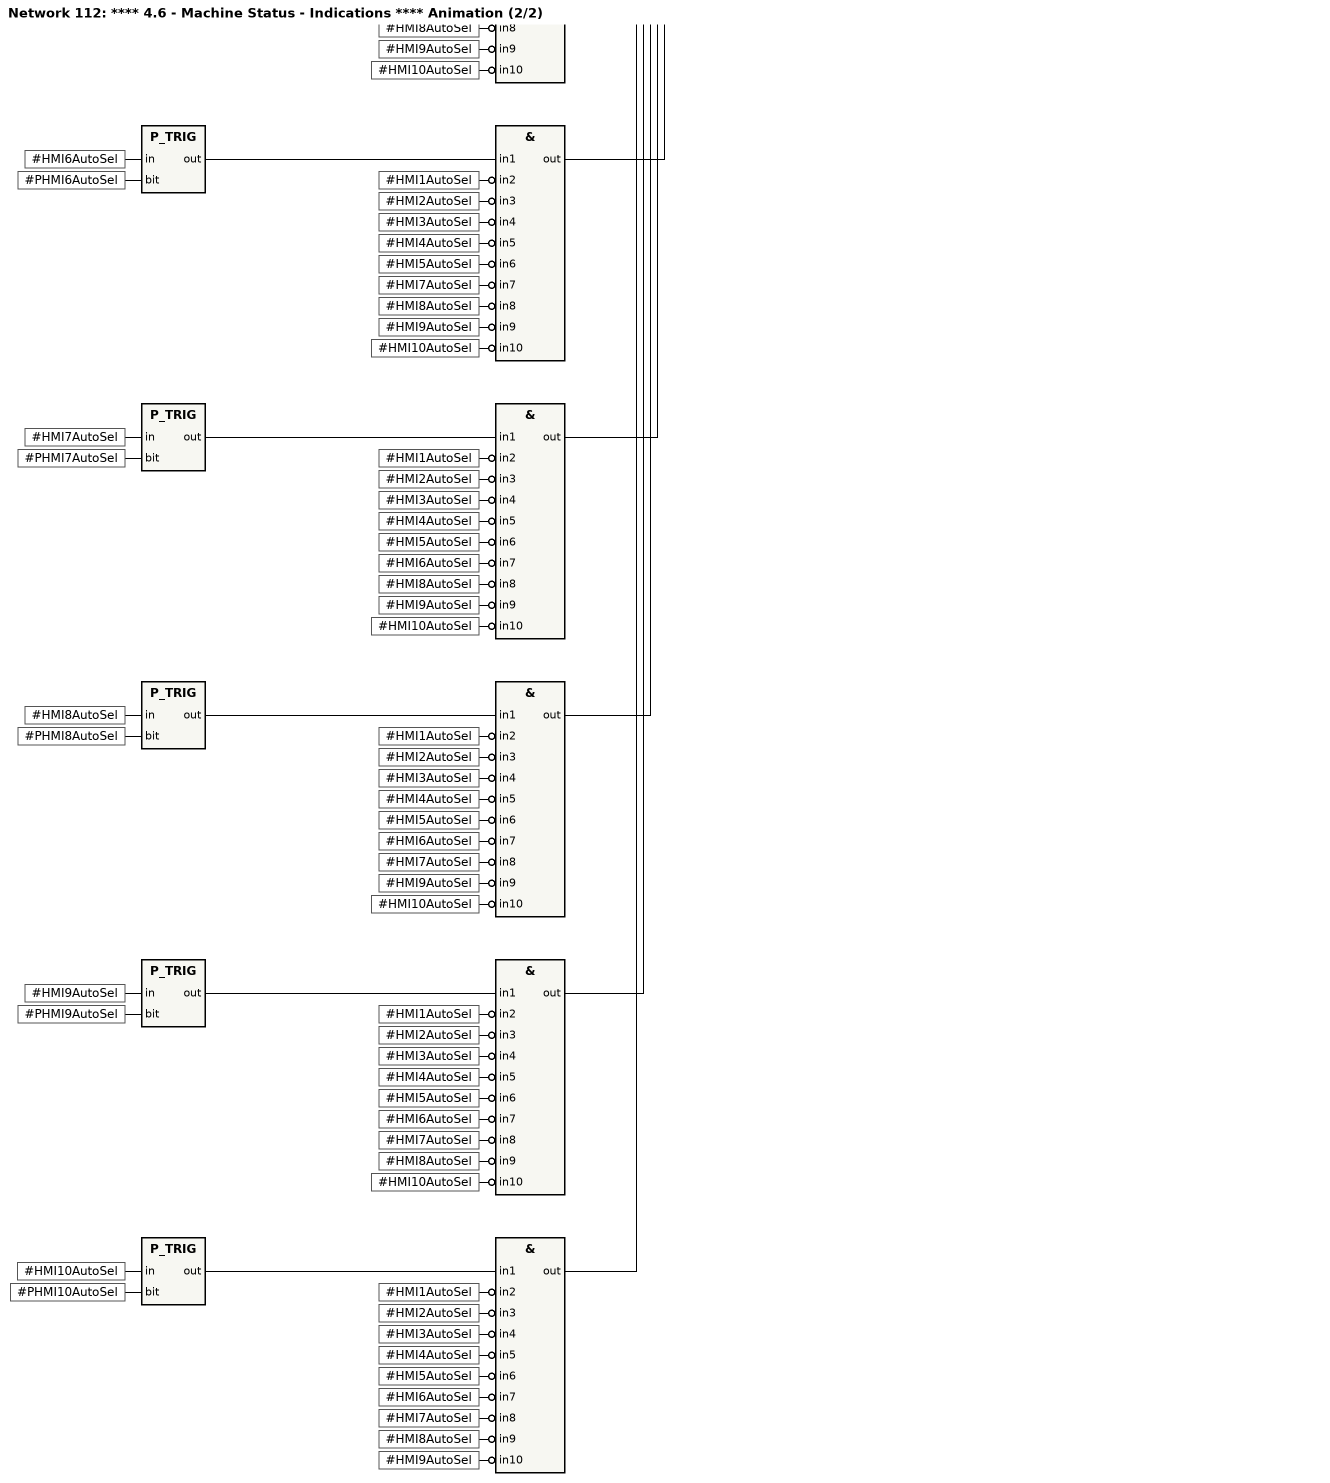
   #_w1 := #HMI1AutoSel AND NOT #PHMI1AutoSel;   // rising edge
   #PHMI1AutoSel := #HMI1AutoSel;
   #_w2 := #HMI2AutoSel AND NOT #PHMI2AutoSel;   // rising edge
   #PHMI2AutoSel := #HMI2AutoSel;
   #_w3 := #HMI3AutoSel AND NOT #PHMI3AutoSel;   // rising edge
   #PHMI3AutoSel := #HMI3AutoSel;
   #_w4 := #HMI4AutoSel AND NOT #PHMI4AutoSel;   // rising edge
   #PHMI4AutoSel := #HMI4AutoSel;
   #_w5 := #HMI5AutoSel AND NOT #PHMI5AutoSel;   // rising edge
   #PHMI5AutoSel := #HMI5AutoSel;
   #_w6 := #HMI6AutoSel AND NOT #PHMI6AutoSel;   // rising edge
   #PHMI6AutoSel := #HMI6AutoSel;
   #_w7 := #HMI7AutoSel AND NOT #PHMI7AutoSel;   // rising edge
   #PHMI7AutoSel := #HMI7AutoSel;
   #_w8 := #HMI8AutoSel AND NOT #PHMI8AutoSel;   // rising edge
   #PHMI8AutoSel := #HMI8AutoSel;
   #_w9 := #HMI9AutoSel AND NOT #PHMI9AutoSel;   // rising edge
   #PHMI9AutoSel := #HMI9AutoSel;
   #_w10 := #HMI10AutoSel AND NOT #PHMI10AutoSel;   // rising edge
   #PHMI10AutoSel := #HMI10AutoSel;
   IF "TRUE" THEN
       "LBitToWord"(I_0 := #HMI1AutoSel AND #HMI2AutoSel AND #HMI3AutoSel AND #HMI4AutoSel AND #HMI5AutoSel AND #HMI6AutoSel AND #HMI7AutoSel AND #HMI8AutoSel AND #HMI9AutoSel AND #HMI10AutoSel,
                    I_1 := (#_w1 AND NOT #HMI2AutoSel AND NOT #HMI3AutoSel AND NOT #HMI4AutoSel AND NOT #HMI5AutoSel AND NOT #HMI6AutoSel AND NOT #HMI7AutoSel AND NOT #HMI8AutoSel AND NOT #HMI9AutoSel AND NOT #HMI10AutoSel) OR (#_w2 AND NOT #HMI1AutoSel AND NOT #HMI3AutoSel AND NOT #HMI4AutoSel AND NOT #HMI5AutoSel AND NOT #HMI6AutoSel AND NOT #HMI7AutoSel AND NOT #HMI8AutoSel AND NOT #HMI9AutoSel AND NOT #HMI10AutoSel) OR (#_w3 AND NOT #HMI1AutoSel AND NOT #HMI2AutoSel AND NOT #HMI4AutoSel AND NOT #HMI5AutoSel AND NOT #HMI6AutoSel AND NOT #HMI7AutoSel AND NOT #HMI8AutoSel AND NOT #HMI9AutoSel AND NOT #HMI10AutoSel) OR (#_w4 AND NOT #HMI1AutoSel AND NOT #HMI2AutoSel AND NOT #HMI3AutoSel AND NOT #HMI5AutoSel AND NOT #HMI6AutoSel AND NOT #HMI7AutoSel AND NOT #HMI8AutoSel AND NOT #HMI9AutoSel AND NOT #HMI10AutoSel) OR (#_w5 AND NOT #HMI1AutoSel AND NOT #HMI2AutoSel AND NOT #HMI3AutoSel AND NOT #HMI4AutoSel AND NOT #HMI6AutoSel AND NOT #HMI7AutoSel AND NOT #HMI8AutoSel AND NOT #HMI9AutoSel AND NOT #HMI10AutoSel) OR (#_w6 AND NOT #HMI1AutoSel AND NOT #HMI2AutoSel AND NOT #HMI3AutoSel AND NOT #HMI4AutoSel AND NOT #HMI5AutoSel AND NOT #HMI7AutoSel AND NOT #HMI8AutoSel AND NOT #HMI9AutoSel AND NOT #HMI10AutoSel) OR (#_w7 AND NOT #HMI1AutoSel AND NOT #HMI2AutoSel AND NOT #HMI3AutoSel AND NOT #HMI4AutoSel AND NOT #HMI5AutoSel AND NOT #HMI6AutoSel AND NOT #HMI8AutoSel AND NOT #HMI9AutoSel AND NOT #HMI10AutoSel) OR (#_w8 AND NOT #HMI1AutoSel AND NOT #HMI2AutoSel AND NOT #HMI3AutoSel AND NOT #HMI4AutoSel AND NOT #HMI5AutoSel AND NOT #HMI6AutoSel AND NOT #HMI7AutoSel AND NOT #HMI9AutoSel AND NOT #HMI10AutoSel) OR (#_w9 AND NOT #HMI1AutoSel AND NOT #HMI2AutoSel AND NOT #HMI3AutoSel AND NOT #HMI4AutoSel AND NOT #HMI5AutoSel AND NOT #HMI6AutoSel AND NOT #HMI7AutoSel AND NOT #HMI8AutoSel AND NOT #HMI10AutoSel) OR (#_w10 AND NOT #HMI1AutoSel AND NOT #HMI2AutoSel AND NOT #HMI3AutoSel AND NOT #HMI4AutoSel AND NOT #HMI5AutoSel AND NOT #HMI6AutoSel AND NOT #HMI7AutoSel AND NOT #HMI8AutoSel AND NOT #HMI9AutoSel),
                    I_2 := #AllHmiAutoSel AND NOT #HMI1LockManual AND NOT #HMI2LockManual AND NOT #HMI3LockManual AND NOT #HMI4LockManual AND NOT #HMI5LockManual AND NOT #HMI6LockManual AND NOT #HMI7LockManual AND NOT #HMI8LockManual AND NOT #HMI9LockManual AND NOT #HMI10LockManual,
                    I_3 := #HMI1LockManual OR #HMI2LockManual OR #HMI3LockManual OR #HMI4LockManual OR #HMI5LockManual OR #HMI6LockManual OR #HMI7LockManual OR #HMI8LockManual OR #HMI9LockManual OR #HMI10LockManual,
                    I_4 := (60 > 0) AND #LockManualTimeout,
                    I_5 := #I_NumHMI > 1,
                    I_6 := "FALSE",
                    I_7 := "FALSE",
                    I_8 := "FALSE",
                    I_9 := "FALSE",
                    I_10 := "FALSE",
                    I_11 := "FALSE",
                    I_12 := "FALSE",
                    I_13 := "FALSE",
                    I_14 := "FALSE",
                    I_15 := #CheckHMIActive,
                    O_Word => #H_Anim);
   END_IF;
END_REGION

REGION Network 113: **** 5.2 - Equations - Flow **** Reset transport memory on active HMI
   // Reset transport memory on active HMI
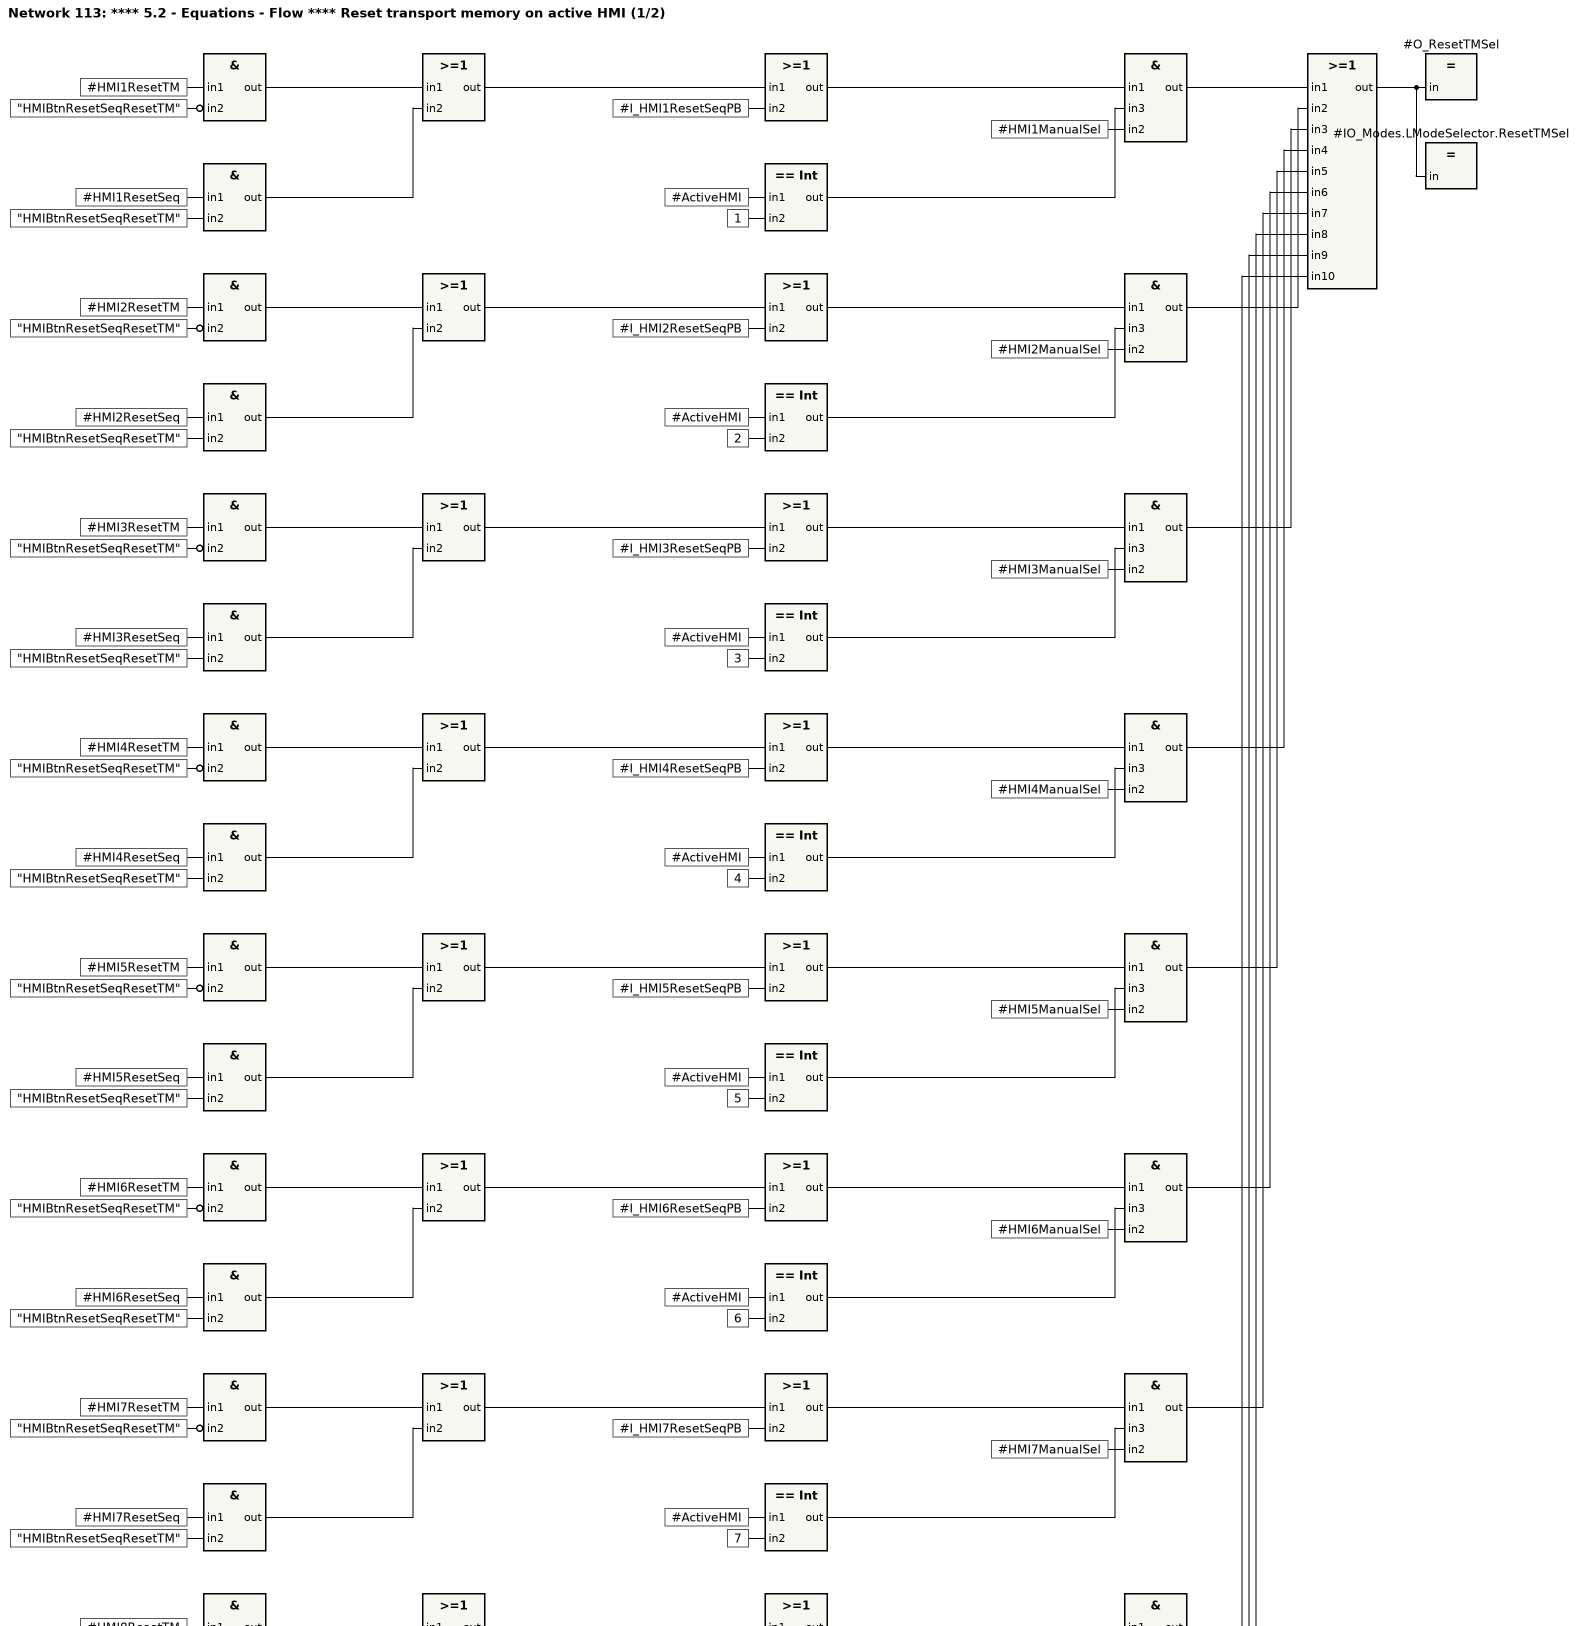
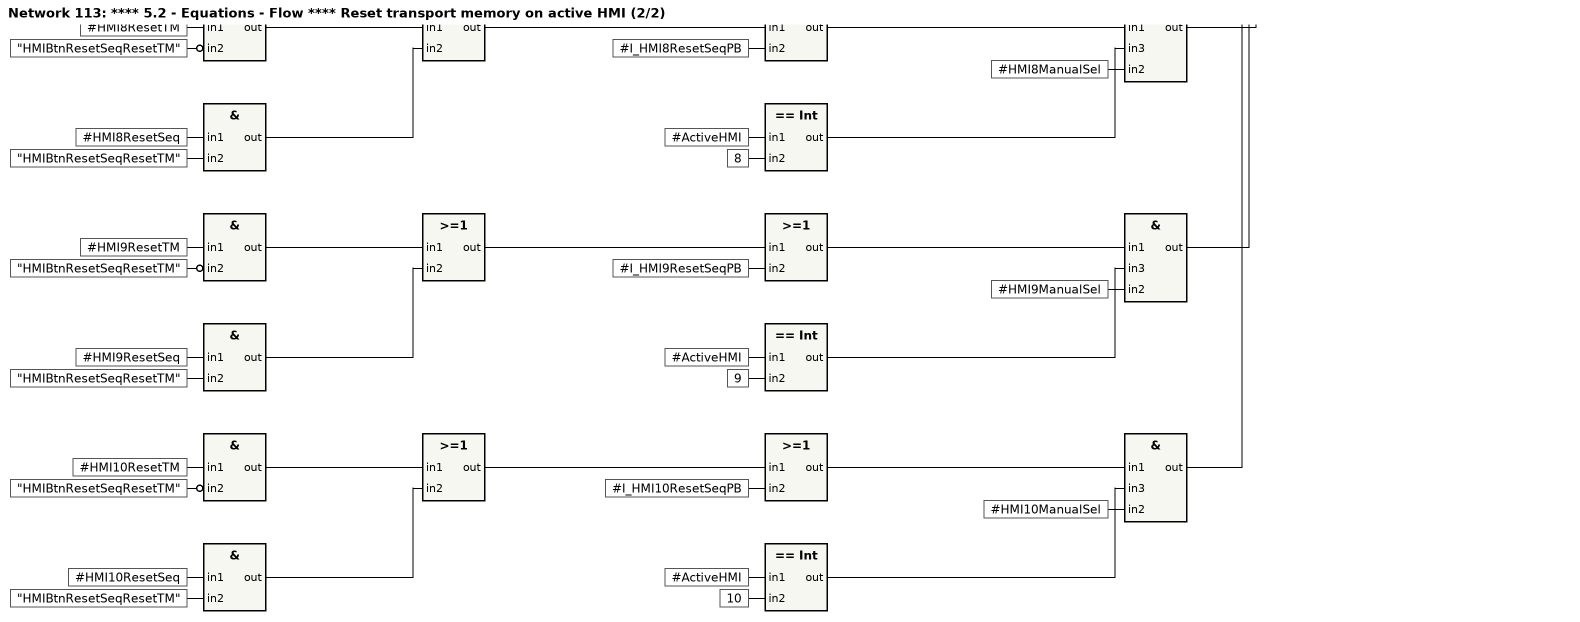
   #O_ResetTMSel := (((#HMI1ResetTM AND NOT "HMIBtnResetSeqResetTM") OR (#HMI1ResetSeq AND "HMIBtnResetSeqResetTM") OR #I_HMI1ResetSeqPB) AND (#ActiveHMI = 1) AND #HMI1ManualSel) OR (((#HMI2ResetTM AND NOT "HMIBtnResetSeqResetTM") OR (#HMI2ResetSeq AND "HMIBtnResetSeqResetTM") OR #I_HMI2ResetSeqPB) AND (#ActiveHMI = 2) AND #HMI2ManualSel) OR (((#HMI3ResetTM AND NOT "HMIBtnResetSeqResetTM") OR (#HMI3ResetSeq AND "HMIBtnResetSeqResetTM") OR #I_HMI3ResetSeqPB) AND (#ActiveHMI = 3) AND #HMI3ManualSel) OR (((#HMI4ResetTM AND NOT "HMIBtnResetSeqResetTM") OR (#HMI4ResetSeq AND "HMIBtnResetSeqResetTM") OR #I_HMI4ResetSeqPB) AND (#ActiveHMI = 4) AND #HMI4ManualSel) OR (((#HMI5ResetTM AND NOT "HMIBtnResetSeqResetTM") OR (#HMI5ResetSeq AND "HMIBtnResetSeqResetTM") OR #I_HMI5ResetSeqPB) AND (#ActiveHMI = 5) AND #HMI5ManualSel) OR (((#HMI6ResetTM AND NOT "HMIBtnResetSeqResetTM") OR (#HMI6ResetSeq AND "HMIBtnResetSeqResetTM") OR #I_HMI6ResetSeqPB) AND (#ActiveHMI = 6) AND #HMI6ManualSel) OR (((#HMI7ResetTM AND NOT "HMIBtnResetSeqResetTM") OR (#HMI7ResetSeq AND "HMIBtnResetSeqResetTM") OR #I_HMI7ResetSeqPB) AND (#ActiveHMI = 7) AND #HMI7ManualSel) OR (((#HMI8ResetTM AND NOT "HMIBtnResetSeqResetTM") OR (#HMI8ResetSeq AND "HMIBtnResetSeqResetTM") OR #I_HMI8ResetSeqPB) AND (#ActiveHMI = 8) AND #HMI8ManualSel) OR (((#HMI9ResetTM AND NOT "HMIBtnResetSeqResetTM") OR (#HMI9ResetSeq AND "HMIBtnResetSeqResetTM") OR #I_HMI9ResetSeqPB) AND (#ActiveHMI = 9) AND #HMI9ManualSel) OR (((#HMI10ResetTM AND NOT "HMIBtnResetSeqResetTM") OR (#HMI10ResetSeq AND "HMIBtnResetSeqResetTM") OR #I_HMI10ResetSeqPB) AND (#ActiveHMI = 10) AND #HMI10ManualSel);
   #IO_Modes.LModeSelector.ResetTMSel := #O_ResetTMSel;
END_REGION

REGION Network 114: **** 5.2 - Equations - Flow **** Reset sequence on active HMI
   // Reset sequence on active HMI
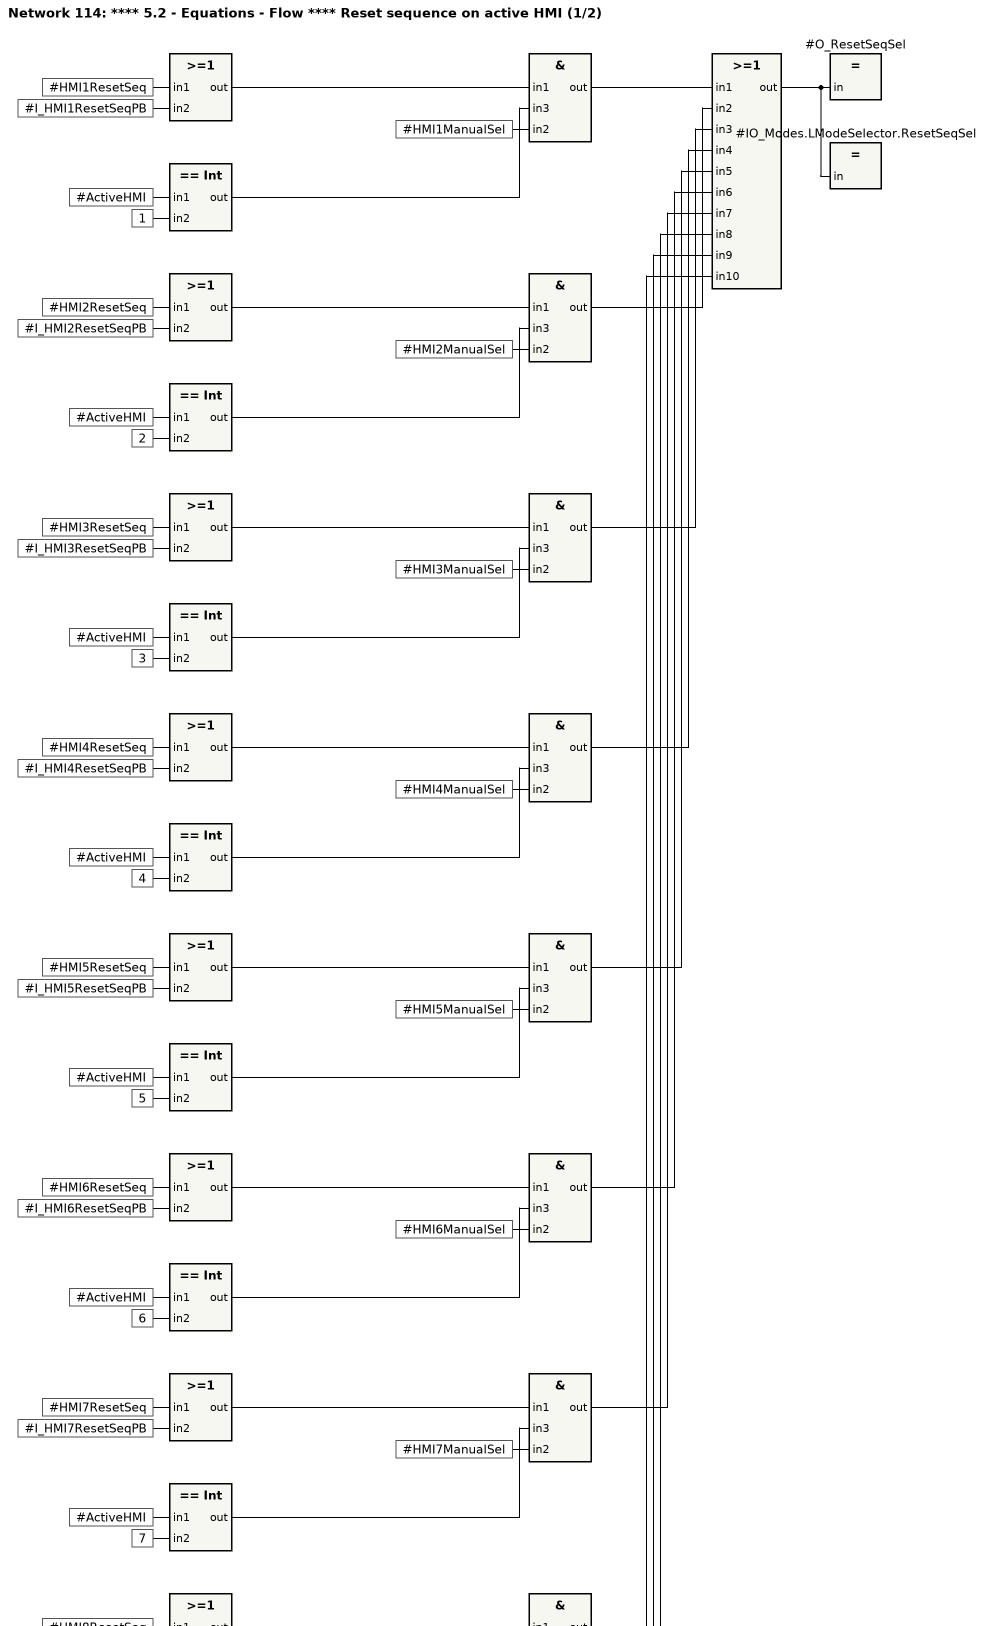
